      global tab_cer_app_g =      [p[0,0,0,0,0,0], p[0,0,0,0,0,0], p[0,0,0,0,0,0], p[0,0,0,0,0,0], p[0,0,0,0,0,0], p[0,0,0,0,0,0], p[0,0,0,0,0,0], p[0,0,0,0,0,0], p[0,0,0,0,0,0], p[0,0,0,0,0,0], p[0,0,0,0,0,0]]
      global tab_cer_deb_g =      [p[0,0,0,0,0,0], p[0,0,0,0,0,0], p[0,0,0,0,0,0], p[0,0,0,0,0,0], p[0,0,0,0,0,0], p[0,0,0,0,0,0], p[0,0,0,0,0,0], p[0,0,0,0,0,0], p[0,0,0,0,0,0], p[0,0,0,0,0,0], p[0,0,0,0,0,0]]
      global tab_cer_quart_g =    [p[0,0,0,0,0,0], p[0,0,0,0,0,0], p[0,0,0,0,0,0], p[0,0,0,0,0,0], p[0,0,0,0,0,0], p[0,0,0,0,0,0], p[0,0,0,0,0,0], p[0,0,0,0,0,0], p[0,0,0,0,0,0], p[0,0,0,0,0,0], p[0,0,0,0,0,0]]
      global tab_cer_mil_g =      [p[0,0,0,0,0,0], p[0,0,0,0,0,0], p[0,0,0,0,0,0], p[0,0,0,0,0,0], p[0,0,0,0,0,0], p[0,0,0,0,0,0], p[0,0,0,0,0,0], p[0,0,0,0,0,0], p[0,0,0,0,0,0], p[0,0,0,0,0,0], p[0,0,0,0,0,0]]
      global tab_cer_tro_g =      [p[0,0,0,0,0,0], p[0,0,0,0,0,0], p[0,0,0,0,0,0], p[0,0,0,0,0,0], p[0,0,0,0,0,0], p[0,0,0,0,0,0], p[0,0,0,0,0,0], p[0,0,0,0,0,0], p[0,0,0,0,0,0], p[0,0,0,0,0,0], p[0,0,0,0,0,0]]
      global tab_cer_fin_g =      [p[0,0,0,0,0,0], p[0,0,0,0,0,0], p[0,0,0,0,0,0], p[0,0,0,0,0,0], p[0,0,0,0,0,0], p[0,0,0,0,0,0], p[0,0,0,0,0,0], p[0,0,0,0,0,0], p[0,0,0,0,0,0], p[0,0,0,0,0,0], p[0,0,0,0,0,0]]
      global tab_cer_ret_g =      [p[0,0,0,0,0,0], p[0,0,0,0,0,0], p[0,0,0,0,0,0], p[0,0,0,0,0,0], p[0,0,0,0,0,0], p[0,0,0,0,0,0], p[0,0,0,0,0,0], p[0,0,0,0,0,0], p[0,0,0,0,0,0], p[0,0,0,0,0,0], p[0,0,0,0,0,0]]

       #2 nouveaux tableaux modif V2.1 (longueur 40 si 4(type)*10(nb soudures max par type) ) -> mis 45 (permettre décalage + marge)
      global tab_type_g = [0,0,0,0,0,0,0,0,0,0,0,0,0,0,0,0,0,0,0,0,0,0,0,0,0,0,0,0,0,0,0,0,0,0,0,0,0,0,0,0,0,0,0,0,0]
      global tab_job_g  = [0,0,0,0,0,0,0,0,0,0,0,0,0,0,0,0,0,0,0,0,0,0,0,0,0,0,0,0,0,0,0,0,0,0,0,0,0,0,0,0,0,0,0,0,0]

      #vitesses de soudure
      global tps_point_g = 0
      global vit_arc_g = [0,0,0,0,0,0,0,0,0,0,0]
      global vit_cer_g = [0,0,0,0,0,0,0,0,0,0,0]
      global vit_lin_g = [0,0,0,0,0,0,0,0,0,0,0]

      global nb_soud_point_g  = 0
      global nb_soud_lin_g    = 0
      global nb_soud_arc_g    = 0
      global nb_soud_cer_g    = 0

      global nbSoudure_glo_g  = 0
  end
  $ 19 "Demande"
  $ 20 "Script: demande_d.script"
  def fun_demande_d():

      close_popup()
      nb_soud_point_d = fun_demande(1)
      if (nb_soud_point_d > 0):
              tps_point_d = request_float_from_primary_client("temps des soudures points ? (s)")
      end
      nb_soud_lin_d = fun_demande(2)
      nb_soud_arc_d = fun_demande(3)
      nb_soud_cer_d = fun_demande(4)

  end
  $ 21 "Script: demande_g.script"
  def fun_demande_g():
       close_popup()
       nb_soud_point_g = fun_demande(1)
       nb_soud_lin_g = fun_demande(2)
       if nb_soud_lin_g > 0:
            vit_lin_g = fun_demande_vit(2)
       end
       nb_soud_arc_g = fun_demande(3)
       if nb_soud_arc_g > 0:
            vit_arc_g = fun_demande_vit(3)
       end
       nb_soud_cer_g = fun_demande(4)
       if nb_soud_arc_g > 0:
            vit_cer_g = fun_demande_vit(4)
       end
  end
  $ 22 "Configuration"
  $ 23 "Script: config_d.script"
  def fun_config_d():

      teach_mode()

          ################### RAZ_des_tableaux ###########################################

      fun_raz_d()

              # Init des variables de traitement
      local type = 0
      local index_soudure_point = 1
      local index_soudure_lin = 1
      local index_soudure_arc = 1
      local index_soudure_cer = 1

      local nbSoudures = 0
      local ajout = False
      close_popup()
      type = fun_demande_type_soudure()
      sync()
      while (type != 5):
          sync()
          if (type == 1):
              if (nb_soud_point_d <10):
                  ajout = True
                  fun_config_soudure_point(index_soudure_point,2) #  le ( ,2) indique la table de droite
                  index_soudure_point = index_soudure_point +1
              else:
                  ajout = False
                  popUp_tropSoudures()
              end

          elif (type == 2):
              if (nb_soud_lin_d <10):
                  ajout = True
                  fun_config_soudure_lineaire(index_soudure_lin,2)
                  index_soudure_lin = index_soudure_lin +1
              else:
                  ajout = False
                  popUp_tropSoudures()
              end

          elif (type == 3):
              if (nb_soud_arc_d <10):
                  ajout = True
                  fun_config_soudure_arc(index_soudure_arc,2)
                  index_soudure_arc = index_soudure_arc +1
              else:
                  ajout = False
                  popUp_tropSoudures()
              end

          elif (type ==4):
              if (nb_soud_cer_d <10):
                  ajout = True
                  fun_config_soudure_cercle(index_soudure_cer,2)
                  index_soudure_cer = index_soudure_cer +1
              else:
                  ajout = False
                  popUp_tropSoudures()
              end

          end

          if (ajout == True):
              tab_type_d[nbSoudures] = type
              tab_job_d[nbSoudures] = fun_demande_job(type)
              nbSoudures = nbSoudures +1
          end

          sync()
          type = fun_demande_type_soudure()
      end
      end_teach_mode()
      global nbSoudure_glo_d = nbSoudures
  end

  $ 24 "Script: config_g.script"
  def fun_config_g():

     teach_mode()

  ######################## Initialisation #######################################

      fun_raz_g()


              # Init des variables de traitement
      local type = 0
      local index_soudure_point = 1
      local index_soudure_lin = 1
      local index_soudure_arc = 1
      local index_soudure_cer = 1

      local nbSoudures = 0
      local ajout = False
      close_popup()
      type = fun_demande_type_soudure()
      sync()
      while (type != 5):
          sync()
          if (type == 1):
              if (nb_soud_point_g <10):
                  ajout = True
                  fun_config_soudure_point(index_soudure_point,1) # ( ,1 indique la table de gauche)
                  index_soudure_point = index_soudure_point +1
              else:
                  ajout = False
                  popUp_tropSoudures()
              end

          elif (type == 2):
              if (nb_soud_lin_g <10):
                  ajout = True
                  fun_config_soudure_lineaire(index_soudure_lin,1)
                  index_soudure_lin = index_soudure_lin +1
              else:
                  ajout = False
                  popUp_tropSoudures()
              end

          elif (type == 3):
              if (nb_soud_arc_g <10):
                  ajout = True
                  fun_config_soudure_arc(index_soudure_arc,1)
                  index_soudure_arc = index_soudure_arc +1
              else:
                  ajout = False
                  popUp_tropSoudures()
              end

          elif (type ==4):
              if (nb_soud_cer_g <10):
                  ajout = True
                  fun_config_soudure_cercle(index_soudure_cer,1)
                  index_soudure_cer = index_soudure_cer +1
              else:
                  ajout = False
                  popUp_tropSoudures()
              end
          end

          if (ajout == True):
              tab_type_g[nbSoudures] = type
              tab_job_g[nbSoudures] = fun_demande_job(type)
              nbSoudures = nbSoudures +1

          end

          sync()
          type = fun_demande_type_soudure()
      end

     end_teach_mode()
     global nbSoudure_glo_g = nbSoudures
  end
  $ 25 "Script: fun_config_soudure_arc.script"
  def fun_config_soudure_arc(index,table):
      if(table == 1):  # sur la table de gauche

          fun_popup_soud(1, 3, index)
          fun_front_up(adresse_bp_cobot)
          tab_arc_app_g[index] =  get_actual_tcp_pose() 	#Enregistrer position dans tableau d approche des soudures arc de cercle quand appui Bp_cobot
          close_popup()

          fun_popup_soud(2, 3, index)
          fun_front_up(adresse_bp_cobot)
          tab_arc_deb_g[index] =  get_actual_tcp_pose() 	#Enregistrer position dans tableau debut quand appui Bp_d
          close_popup()

          fun_popup_soud(4, 3, index)
          fun_front_up(adresse_bp_cobot)
          tab_arc_mil_g[index] =  get_actual_tcp_pose() 	#Enregistrer position dans tableau milieu quand appui Bp_cobot
          close_popup()

          fun_popup_soud(6, 3, index)
          fun_front_up(adresse_bp_cobot)
          tab_arc_fin_g[index] =  get_actual_tcp_pose() 	#Enregistrer position dans un tableau fin quand appui Bp_cobot
          close_popup()

          vit_arc_g[index] = fun_demande_vit(3)           #demande de vitesse des soudures lineaire

          fun_popup_soud(7, 3, index)
          fun_front_up(adresse_bp_cobot)
          tab_arc_ret_g[index] =  get_actual_tcp_pose() 	#Enregistrer position dans tableau retrait quand appui Bp_cobot
          close_popup()

          nb_soud_arc_g = nb_soud_arc_g +1

      else: #sur la table de droite
          fun_popup_soud(1, 3, index)
          fun_front_up(adresse_bp_cobot)
          tab_arc_app_d[index] =  get_actual_tcp_pose() 	#Enregistrer position dans tableau d approche des soudures arc de cercle quand appui Bp_cobot
          close_popup()

          fun_popup_soud(2, 3, index)
          fun_front_up(adresse_bp_cobot)
          tab_arc_deb_d[index] =  get_actual_tcp_pose() 	#Enregistrer position dans tableau debut quand appui Bp_d
          close_popup()

          fun_popup_soud(4, 3, index)
          fun_front_up(adresse_bp_cobot)
          tab_arc_mil_d[index] =  get_actual_tcp_pose() 	#Enregistrer position dans tableau milieu quand appui Bp_cobot
          close_popup()

          fun_popup_soud(6, 3, index)
          fun_front_up(adresse_bp_cobot)
          tab_arc_fin_d[index] =  get_actual_tcp_pose() 	#Enregistrer position dans un tableau fin quand appui Bp_cobot
          close_popup()

          vit_arc_d[index] = fun_demande_vit(3)           #demande de vitesse des soudures lineaire

          fun_popup_soud(7, 3, index)
          fun_front_up(adresse_bp_cobot)
          tab_arc_ret_d[index] =  get_actual_tcp_pose() 	#Enregistrer position dans tableau retrait quand appui Bp_cobot
          close_popup()

          nb_soud_arc_d = nb_soud_arc_d +1
      end
  end
  $ 26 "Script: fun_config_soudure_cercle.script"
  def fun_config_soudure_cercle(index,table):
      if(table == 1):  # sur la table de gauche

          fun_popup_soud(1, 4, index)
          fun_front_up(adresse_bp_cobot)
          tab_cer_app_g[index] =  get_actual_tcp_pose()     	#Enregistrer position dans tableau d approche des soudures arc de cercle quand appui Bp_cobot
          close_popup()

          fun_popup_soud(2, 4, index)
          fun_front_up(adresse_bp_cobot)
          tab_cer_deb_g[index] =  get_actual_tcp_pose()     	#Enregistrer position dans tableau debut quand appui Bp_cobot
          close_popup()

          fun_popup_soud(3, 4, index)
          fun_front_up(adresse_bp_cobot)
          tab_cer_quart_g[index] =  get_actual_tcp_pose()   	#Enregistrer position dans tableau d'approche des soudures arc de cercle quand appui Bp_d
          close_popup()

          fun_popup_soud(4, 4, index)
          fun_front_up(adresse_bp_cobot)
          tab_cer_mil_g[index] =  get_actual_tcp_pose()     	#Enregistrer position dans tableau milieu quand appui Bp_cobot
          close_popup()

          fun_popup_soud(5, 4, index)
          fun_front_up(adresse_bp_cobot)
          tab_cer_tro_g[index] =  get_actual_tcp_pose()     	#Enregistrer position dans tableau milieu quand appui Bp_cobot
          close_popup()

          fun_popup_soud(6, 4, index)
          fun_front_up(adresse_bp_cobot)
          tab_cer_fin_g[index] =  get_actual_tcp_pose()     	#Enregistrer position dans un tableau fin quand appui Bp_cobot
          close_popup()

          vit_cer_g[index] = fun_demande_vit(4)

          fun_popup_soud(7, 4, index)
          fun_front_up(adresse_bp_cobot)
          tab_cer_ret_g[index] =  get_actual_tcp_pose()    	#position de retrait est la meme que position d approche
          close_popup()

          nb_soud_cer_g= nb_soud_cer_g + 1
      else: #sur la table de droite

          fun_popup_soud(1, 4, index)
          fun_front_up(adresse_bp_cobot)
          tab_cer_app_d[index] =  get_actual_tcp_pose()     	#Enregistrer position dans tableau d approche des soudures arc de cercle quand appui Bp_cobot
          close_popup()

          fun_popup_soud(2, 4, index)
          fun_front_up(adresse_bp_cobot)
          tab_cer_deb_d[index] =  get_actual_tcp_pose()     	#Enregistrer position dans tableau debut quand appui Bp_cobot
          close_popup()

          fun_popup_soud(3, 4, index)
          fun_front_up(adresse_bp_cobot)
          tab_cer_quart_d[index] =  get_actual_tcp_pose()   	#Enregistrer position dans tableau d'approche des soudures arc de cercle quand appui Bp_d
          close_popup()

          fun_popup_soud(4, 4, index)
          fun_front_up(adresse_bp_cobot)
          tab_cer_mil_d[index] =  get_actual_tcp_pose()     	#Enregistrer position dans tableau milieu quand appui Bp_cobot
          close_popup()

          fun_popup_soud(5, 4, index)
          fun_front_up(adresse_bp_cobot)
          tab_cer_tro_d[index] =  get_actual_tcp_pose()     	#Enregistrer position dans tableau milieu quand appui Bp_cobot
          close_popup()

          fun_popup_soud(6, 4, index)
          fun_front_up(adresse_bp_cobot)
          tab_cer_fin_d[index] =  get_actual_tcp_pose()     	#Enregistrer position dans un tableau fin quand appui Bp_cobot
          close_popup()

          vit_cer_d[index] = fun_demande_vit(4)

          fun_popup_soud(7, 4, index)
          fun_front_up(adresse_bp_cobot)
          tab_cer_ret_d[index] =  get_actual_tcp_pose()    	#position de retrait est la meme que position d approche
          close_popup()

          nb_soud_cer_d = nb_soud_cer_d +1
      end
  end
  $ 27 "Script: fun_config_soudure_lineaire.script"
  def fun_config_soudure_lineaire(index, table):
      if(table == 1):  # sur la table de gauche

          fun_popup_soud(1, 2, index)
          fun_front_up(adresse_bp_cobot)
          tab_lin_app_g[index] =  get_actual_tcp_pose()     	#Enregistrer position dans tableau d approche des soudures lineaire quand appui Bp_cobot
          close_popup()

          fun_popup_soud(2, 2, index)
          fun_front_up(adresse_bp_cobot)
          tab_lin_deb_g[index] =  get_actual_tcp_pose()     	#Enregistrer position dans tableau debut quand appui Bp_cobot
          close_popup()

          fun_popup_soud(6, 2, index)
          fun_front_up(adresse_bp_cobot)
          tab_lin_fin_g[index] =  get_actual_tcp_pose()     	#Enregistrer position dans un tableau fin quand appui Bp_cobot
          close_popup()

          vit_lin_g[index] = fun_demande_vit(2)

          fun_popup_soud(7, 2, index)
          fun_front_up(adresse_bp_cobot)
          tab_lin_ret_g[index] =  get_actual_tcp_pose()     	#Enregistrer position dans tableau retrait quand appui Bp_cobot
          close_popup()

          nb_soud_lin_g = nb_soud_lin_g +1

      else: #sur la table de droite

          fun_popup_soud(1, 2, index)
          fun_front_up(adresse_bp_cobot)
          tab_lin_app_d[index] =  get_actual_tcp_pose()     	#Enregistrer position dans tableau d approche des soudures lineaire quand appui Bp_cobot
          close_popup()

          fun_popup_soud(2, 2, index)
          fun_front_up(adresse_bp_cobot)
          tab_lin_deb_d[index] =  get_actual_tcp_pose()     	#Enregistrer position dans tableau debut quand appui Bp_cobot
          close_popup()

          fun_popup_soud(6, 2, index)
          fun_front_up(adresse_bp_cobot)
          tab_lin_fin_d[index] =  get_actual_tcp_pose()     	#Enregistrer position dans un tableau fin quand appui Bp_cobot
          close_popup()

          vit_lin_d[index] = fun_demande_vit(2)

          fun_popup_soud(7, 2, index)
          fun_front_up(adresse_bp_cobot)
          tab_lin_ret_d[index] =  get_actual_tcp_pose()     	#Enregistrer position dans tableau retrait quand appui Bp_cobot
          close_popup()

          nb_soud_lin_d = nb_soud_lin_d +1
      end
  end
  $ 28 "Script: fun_config_soudure_point.script"
  def fun_config_soudure_point(index,table):

      if(table == 1):  # sur la table de gauche


          fun_popup_soud(1, 1, index)
          fun_front_up(adresse_bp_cobot)
          tab_point_app_g[index] =  get_actual_tcp_pose()   #Enregistrer position dans tableau d'approche des soudue points quand appui bouton
          close_popup()

          fun_popup_soud(2, 1, index)
          fun_front_up(adresse_bp_cobot)
          tab_point_deb_g[index] =  get_actual_tcp_pose()   #Enregistrer position debut quand appui bouton bp_cobot
          close_popup()

          tab_point_ret_g[index] = tab_point_app_g[index]         #point de retrait est le meme que le point d approche

          nb_soud_point_g = nb_soud_point_g +1

          if (nb_soud_point_g <= 1 ):
              tps_point_g = request_float_from_primary_client("temps des soudures points ? (s)")
          end




          sync()
      else: #sur la table de droite

          fun_popup_soud(1, 1, index)
          fun_front_up(adresse_bp_cobot)
          tab_point_app_d[index] =  get_actual_tcp_pose()   #Enregistrer position dans tableau d'approche des soudue points quand appui bouton
          close_popup()

          fun_popup_soud(2, 1, index)
          fun_front_up(adresse_bp_cobot)
          tab_point_deb_d[index] =  get_actual_tcp_pose()   #Enregistrer position debut quand appui bouton bp_cobot
          close_popup()

          tab_point_ret_d[index] = tab_point_app_d[index]         #point de retrait est le meme que le point d approche

          nb_soud_point_d = nb_soud_point_d +1

          if (nb_soud_point_d <= 1 ):
              tps_point_d = request_float_from_primary_client("temps des soudures points ? (s)")
          end


          sync()
      end
  end
  $ 29 "Script: popUp_tropSoudures.script"
  def popUp_tropSoudures():
      close_popup()
      popUp_tropSoudures = "Ajout impossible, deja 10 soudures de ce type"
      socket_open("127.0.0.1",29999,"internal") # open internal socket
      socket_send_line(popUp_tropSoudures,"internal")     #Affichage message
      socket_send_byte(10,"internal")
  end
  $ 30 "Script: valid_config_d.script"

  def fun_valid_config_d():
      #on demande la validation de la configuration

      validation_d = request_boolean_from_primary_client("Valider la configuration de la table droite ? Cliquer sur non pour effacer les paramètres.")

          if(validation_d ==True):

              popup2 = "popup La programmation de la pièce droite est terminée."
              socket_open("127.0.0.1",29999,"internal") # open internal socket
              socket_send_line(popup2,"internal")     #Affichage message
              socket_send_byte(10,"internal")
          config_d = 1

          else:
          nb_soud_point_d = 0
          nb_soud_lin_d = 0
          nb_soud_arc_d = 0
          nb_soud_cer_d = 0
          config_d = 0

          fun_raz_d()

          popup3 = "popup La programmation de la pièce droite a été effacée."
          socket_open("127.0.0.1",29999,"internal") # open internal socket
          socket_send_line(popup3,"internal")     #Affichage message
          socket_send_byte(10,"internal")
      end
  end
  $ 31 "Script: valid_config_g.script"
  def fun_valid_config_g():
  #on demande la validation de la configuration

      alidation_g = request_boolean_from_primary_client("Valider la programmation de la table gauche ? Cliquer sur non pour effacer les paramètres.")

      if(validation_g ==True):

          popup2 = "popup La programmation de la pièce gauche est terminée."
          socket_open("127.0.0.1",29999,"internal") # open internal socket
          socket_send_line(popup2,"internal")     #Affichage message
          socket_send_byte(10,"internal")
      config_g =1
      else:

      nb_soud_point_g = 0
      nb_soud_lin_g = 0
      nb_soud_arc_g = 0
      nb_soud_cer_g = 0
      config_g = 0

      fun_raz_g()


      popup3 = "popup La programmation de la pièce gauche a été effacée."
      socket_open("127.0.0.1",29999,"internal") # open internal socket
      socket_send_line(popup3,"internal")     #Affichage message
      socket_send_byte(10,"internal")

      end
  end
  $ 32 "Execution"
  $ 33 "Script: execution_d.script"
  def fun_execution_d():
      ######################## INITIALISATION #########################################
      #adressage
      adresse_bp_cobot = 2                                    #adresse cobot bp_cobot
      adresse_bp_d = 3                                        #adresse cobot bp_g
  #VARIABLES CI DESSUS UTILES ?????


      local index_soudure_point = 1
      local index_soudure_lin = 1
      local index_soudure_arc = 1
      local index_soudure_cer = 1

      close_popup()
      #config popup
      popup1 = "popup Table droite, éxécution..."
      socket_open("127.0.0.1",29999,"internal")
      socket_send_line(popup1,"internal")
      socket_send_byte(10,"internal")

      fun_deplacement_pose_inter(2)    #deplacement dans la position intermédiaire enregistrée

      local nbSoudures = nbSoudure_glo_d
      local soudureEnCours = 0 #soudure en cours
      local job = 0
      local typeSoudure = 0

      while (soudureEnCours<nbSoudures): #pour le moment début a 0 donc < (a voir si changement necessaire)
          job = tab_job_d[soudureEnCours]
          fun_commande_job(job)
          typeSoudure = tab_type_d[soudureEnCours]

          #switch de tous les types avec appel aux fonctions correspondantes
          if (typeSoudure == 1 ):
              fun_soudure_point(index_soudure_point,2) # ( , 2 pour signifier table de droite )
              #fun_soudure_point(index_soudure_point)
              index_soudure_point = index_soudure_point + 1
          elif (typeSoudure == 2 ):
              fun_soudure_lineaire(index_soudure_lin,2)
              index_soudure_lin = index_soudure_lin + 1
          elif (typeSoudure == 3 ):
              fun_soudure_arc(index_soudure_arc,2)
              index_soudure_arc = index_soudure_arc +1
          elif (typeSoudure == 4 ):
              fun_soudure_cercle(index_soudure_cercle,2)
              index_soudure_cercle = index_soudure_cercle +1
          else:
          end
          soudureEnCours = soudureEnCours +1
          sync()
      end
          #movej(anti_poq_d_1, a=1.4,v=1.1,t=0,r=0.005)
          #movej(anti_poq_d_2, a=1.4,v=1.1,t=0,r=0.005)
          movej(Point_Attente_D, a=0.8,v=1.05,t=0,r=0.005)
          movej(Point_init_D, a=0.8,v=1.05,t=0,r=0.005)
          movej(Point_avt_initD, a=0.8,v=1.05,t=0,r=0.005)
          movej(Point_init, a=0.8,v=1.05,t=0,r=0)
  end
  $ 34 "Script: execution_g.script"
  def fun_execution_g():
  ######################## INITIALISATION #######################################

  #adressage
  adresse_bp_cobot = 2                                    #adresse cobot bp_cobot
  adresse_bp_g = 2                                        #adresse cobot bp_g
  #VARIABLES CI DESSUS UTILES ?????


  local index_soudure_point = 1
  local index_soudure_lin = 1
  local index_soudure_arc = 1
  local index_soudure_cer = 1

  close_popup()
  #config popup
  #popup1 = "popup Table gauche, éxécution..."
  #socket_open("127.0.0.1",29999,"internal")
  #socket_send_line(popup1,"internal")
  #socket_send_byte(10,"internal")

  #fun_deplacement_pose_inter(1)

  local nbSoudures = nbSoudure_glo_g
  local soudureEnCours = 0 #soudure en cours
  local job = 0
  local typeSoudure = 0

  while (soudureEnCours<nbSoudures): #pour le moment début a 0 donc < (a voir si changement necessaire)
      job = tab_job_g[soudureEnCours]
      fun_commande_job(job)
      typeSoudure = tab_type_g[soudureEnCours]

      #switch de tous les types avec appel aux fonctions correspondantes
      if (typeSoudure == 1 ):
          #fun_soudure_point(index_soudure_point)
          fun_soudure_point(index_soudure_point,1) # ( , 1 pour signifier table de gauche )
          index_soudure_point = index_soudure_point + 1
      elif (typeSoudure == 2 ):
          fun_soudure_lineaire(index_soudure_lin,1)
          index_soudure_lin = index_soudure_lin + 1
      elif (typeSoudure == 3 ):
          fun_soudure_arc(index_soudure_arc,1)
          index_soudure_arc = index_soudure_arc +1
      elif (typeSoudure == 4 ):
          fun_soudure_cercle(index_soudure_cercle,1)
          index_soudure_cercle = index_soudure_cercle +1
      else:
      end
      soudureEnCours = soudureEnCours +1
      sync()
  end
      #movej(anti_Poq_g, a=1.4,v=1.1,t=0,r=0.005)
      #movej(Point_init, a=1.4,v=1.1,t=0,r=0.005)

     # movej(Point_Attente_G, a=0.8,v=1.05,t=0,r=0.005)
      #movej(Point_init_G, a=0.8,v=1.05,t=0,r=0.005)
     # movej(Point_init, a=0.8,v=1.05,t=0,r=0)

  end
  $ 35 "Script: fun_activer_soudure.script"
  def fun_activer_soudure():
      soudure_on = 1
      sleep(tps_init_soud)
      sync()
  end
  $ 36 "Script: fun_fin_soudure.script"
  def fun_fin_soudure(table):

      soudure_on = 0
      while(fin_soud == 0):
      end
      set_digital_out(table+4,False)                 #eteindre la lumiere pour dire que l'on soude plus

      #table +4 : les sorties numériques sont respectivements 5 table gauche & 6 table droite
      #le décalage permet d'écrire directement au bon endroit
      sync()

  end
  $ 37 "Script: fun_commande_job.script"
  #fonction ecriture des jobs vers rob3000
  def fun_commande_job(int):

      if (int == 0):
          set_digital_out(2,False)
          set_digital_out(3,False)


      elif(int == 1):
          set_digital_out(2,True)
          set_digital_out(3,False)

      elif(int == 2):
          set_digital_out(2,False)
          set_digital_out(3,True)

      elif(int == 3):
          set_digital_out(2,True)
          set_digital_out(3,True)

     # else:
     #     set_digital_out(2,False)
       #   set_digital_out(3,False)
      end
  end
  $ 38 "Script: fun_deplacement_pose_inter.script"
  def fun_deplacement_pose_inter(table):
      a_fun = 0.2
      v_fun = 1.1
      r_fun= 0
      t_fun = 0
      if (table == 1): #si 1 -> Table de gauche
        #  movej(pose_inter_g,a=a_fun,v=v_fun,t=t_fun,r=r_fun)
      else: #sinon table de droite
       #   movej(pose_inter_d,a=a_fun,v=v_fun,t=t_fun,r=r_fun)
      end
      sync()
  end
  $ 39 "Script: fun_soudure_arc.script"
  def fun_soudure_arc(Index,table):
      a_fun = 0.5
      v_fun = 1.1
      r_fun= 0.00
      t_fun = 0
      if (table == 1): #si 1 -> Table de gauche

          movej(tab_arc_app_g[Index],a_fun,v=v_fun,t=t_fun,r=r_fun)
          set_digital_out(5,True)                     #Allumer la lumiere pour dire que l'on soude
          movej(tab_arc_deb_g[Index],a_fun,v=v_fun,t=t_fun,r=r_fun)

          fun_activer_soudure()                        #appel de la fonction activer la soudure

          movec(tab_arc_mil_g[Index], tab_arc_fin_g[Index], a_fun,v=vit_arc_g[Index], r=0.002)

          fun_fin_soudure(1)                           #appel de la fonction désactiver la soudure

          movej(tab_arc_ret_g[Index],a=a_fun,v=v_fun,t=t_fun,r=r_fun)

          fun_deplacement_pose_inter(1)                     #appel de la fonction de déplacement en pose intermédiaire

      else: #sinon table de droite

          movej(tab_arc_app_d[Index],a_fun,v=v_fun,t=t_fun,r=r_fun)
          set_digital_out(6,True)                     #Allumer la lumiere pour dire que l'on soude
          movej(tab_arc_deb_d[Index],a_fun,v=v_fun,t=t_fun,r =r_fun)

          fun_activer_soudure()                        #appel de la fonction activer la soudure

          movec(tab_arc_mil_d[Index], tab_arc_fin_d[Index], a_fun,v=vit_arc_d[Index], r=0.002)

          fun_fin_soudure(2)                           #appel de la fonction désactiver la soudure

          movej(tab_arc_ret_d[Index],a_fun,v=v_fun,t=t_fun,r=r_fun)

          fun_deplacement_pose_inter(2)                     #appel de la fonction de déplacement en pose intermédiaire
      end
      sync()
  end
  $ 40 "Script: fun_soudure_cercle.script"
  def fun_soudure_cercle(Index,table):
      a_fun = 0.5
      v_fun = 1.1
      r_fun= 0.0
      t_fun = 0
      if (table == 1): #si 1 -> Table de gauche
          movej(tab_cer_app_g[Index],a=a_fun,v=v_fun,t=t_fun,r=r_fun)
          set_digital_out(5,True)                     #Allumer la lumiere pour dire que l'on soude
          movej(tab_cer_deb_g[Index],a=a_fun,v=v_fun,t=t_fun,r=r_fun)

          fun_activer_soudure()                        #appel de la fonction activer la soudure

          movec(tab_cer_quart_g[Index], tab_cer_mil_g[Index], a=a_fun,v=vit_cer_g[Index], r=0.002)
          movec(tab_cer_tro_g[Index], tab_cer_fin_g[Index], a=a_fun,v=vit_cer_g[Index], r=0.002)

          fun_fin_soudure(1)                           #appel de la fonction désactiver la soudure

          movej(tab_cer_ret_g[Index],a=a_fun, v=v_fun, t=t_fun, r=r_fun)

          fun_deplacement_pose_inter(1)                     #appel de la fonction de déplacement en pose intermédiaire

      else: #sinon table de droite
          movej(tab_cer_app_d[Index],a=a_fun,v=v_fun,t=t_fun,r=r_fun)
          set_digital_out(6,True)                     #Allumer la lumiere pour dire que l'on soude
          movej(tab_cer_deb_d[Index],a=a_fun,v=v_fun,t=t_fun,r=r_fun)

          fun_activer_soudure()                       #appel de la fonction activer la soudure

          movec(tab_cer_quart_d[Index], tab_cer_mil_d[Index], a=a_fun,v=vit_cer_d[Index], r=0.002)
          movec(tab_cer_tro_d[Index], tab_cer_fin_d[Index], a=a_fun, v=vit_cer_d[Index], r=0.002)

          fun_fin_soudure(2)                           #appel de la fonction désactiver la soudure

          movej(tab_cer_ret_d[Index],a=a_fun, v=v_fun, t=t_fun, r=r_fun)

          fun_deplacement_pose_inter(2)                     #appel de la fonction de déplacement en pose intermédiaire

      end
      sync()
  end
  $ 41 "Script: fun_soudure_lineaire.script"
  def fun_soudure_lineaire(Index,table):
      a_fun = 2
      v_fun = 4
      r_fun= 0.00
      t_fun = 0
      if (table == 1): #si 1 -> Table de gauche
          movej(tab_lin_app_g[Index],a=a_fun,v=v_fun,t=t_fun,r=r_fun)
          set_digital_out(5,True)                     #Allumer la lumiere pour dire que l'on soude
          movej(tab_lin_deb_g[Index],a=a_fun,v=v_fun,t=t_fun,r=r_fun)

          fun_activer_soudure()                         #appel de la fonction activer la soudure

          movel(tab_lin_fin_g[Index],a=a_fun,v=vit_lin_g[Index],t=t_fun)

          fun_fin_soudure(1)                           #appel de la fonction désactiver la soudure

          movej(tab_lin_ret_g[Index],a=a_fun,v=v_fun,t=t_fun,r=r_fun)

          fun_deplacement_pose_inter(1)                     #appel de la fonction de déplacement en pose intermédiaire


      else: #sinon table de droite

          movej(tab_lin_app_d[Index],a=a_fun,v=v_fun,t=t_fun,r=r_fun)
          set_digital_out(6,True)                     #Allumer la lumiere pour dire que l'on soude
          movej(tab_lin_deb_d[Index],a=a_fun,v=v_fun,t=t_fun,r=r_fun)

          fun_activer_soudure()                         #appel de la fonction activer la soudure

          movel(tab_lin_fin_d[Index],a=a_fun,v=vit_lin_d[Index],t=t_fun)

          fun_fin_soudure(2)                           #appel de la fonction désactiver la soudure

          movej(tab_lin_ret_d[Index],a=a_fun,v=v_fun,t=t_fun,r=r_fun)

          fun_deplacement_pose_inter(2)                     #appel de la fonction de déplacement en pose intermédiaire

      end
      sync()
  end
  $ 42 "Script: fun_soudure_point.script"
  def fun_soudure_point(Index,table):
      a_fun = 0.5
      v_fun = 1.1
      r_fun= 0.00
      t_fun = 0
      if (table == 1): #si 1 -> Table de gauche
          movej(tab_point_app_g[Index],a=a_fun,v=v_fun,t=t_fun,r= r_fun)
          set_digital_out(5,True)                     #Allumer la lumiere pour dire que l'on soude
          movej(tab_point_deb_g[Index],a=a_fun,v=v_fun,t=t_fun,r= r_fun)

          fun_activer_soudure()                         #appel de la fonction activer la soudure

          sleep(tps_point_g)                          #temps de soudure

          fun_fin_soudure(1)                           #appel de la fonction désactiver la soudure

          movej(tab_point_ret_g[Index],a=a_fun,v=v_fun,t=t_fun,r= r_fun)
          fun_deplacement_pose_inter(1)                     #appel de la fonction de déplacement en pose intermédiaire

      else: #sinon table de droite
          movej(tab_point_app_d[Index],a=a_fun,v=v_fun,t=t_fun,r= r_fun)
          set_digital_out(6,True)                     #Allumer la lumiere pour dire que l'on soude
          movej(tab_point_deb_d[Index],a=a_fun,v=v_fun,t=t_fun,r= r_fun)

          fun_activer_soudure()                         #appel de la fonction activer la soudure

          sleep(tps_point_d)                          #temps de soudure

          fun_fin_soudure(2)                           #appel de la fonction désactiver la soudure

          movej(tab_point_ret_d[Index],a=a_fun,v=v_fun,t=t_fun,r=r_fun)
          fun_deplacement_pose_inter(2)                     #appel de la fonction de déplacement en pose intermédiaire

      end
      sync()
  end
  $ 43 "Pas_A_Pas"
  $ 44 "Script: fun_ajouter_soudure.script"
  def fun_ajouter_soudure(sens,soudureEnCours, index_soudure_point, index_soudure_lin,index_soudure_arc,index_soudure_cercle,table):
      #pour le moment pas de vérif de trop de mouvements (doit etre inferiruer à 9par par type)

      if (table ==1):
          nbSoudures = nbSoudure_glo_g
      elif(table ==2):
          nbSoudures = nbSoudure_glo_d
      end
      local nbDecalage = 0
      local index = soudureEnCours
      local typeSoudure = 0
      local nb_soudure_type = 0
      typeSoudure = fun_demande_type_soudure()

      if (typeSoudure == 1):
        indexTypeSoudure = index_soudure_point
        if (table ==1):
            nb_soudure_type = nb_soud_point_g
        elif(table ==2):
            nb_soudure_type = nb_soud_point_d
        end
      elif (typeSoudure == 2):
          indexTypeSoudure = index_soudure_lin
          if (table ==1):
              nb_soudure_type = nb_soud_lin_g
          elif(table ==2):
              nb_soudure_type = nb_soud_lin_d
          end
      elif(typeSoudure == 3):
          indexTypeSoudure = index_soudure_arc
          if (table ==1):
              nb_soudure_type = nb_soud_arc_g
          elif(table ==2):
              nb_soudure_type = nb_soud_arc_d
          end
      elif(typeSoudure == 4):
          indexTypeSoudure = index_soudure_cercle
          if (table ==1):
              nb_soudure_type = nb_soud_cer_g
          elif(table ==2):
              nb_soudure_type = nb_soud_cer_d
          end
      end

      if (sens == 2):  #AJOUTER AVANT


          #pour les tableaux qui type & job
          index_tab_typejob = nbSoudures -1
          while(index_tab_typejob >= soudureEnCours ):
              if (table ==1):
                  tab_job_g[index_tab_typejob +1] = tab_job_g[index_tab_typejob]
                  tab_type_g[index_tab_typejob +1] = tab_type_g[index_tab_typejob]
              else:
                  tab_job_d[index_tab_typejob +1] = tab_job_d[index_tab_typejob]
                  tab_type_d[index_tab_typejob +1] = tab_type_d[index_tab_typejob]
              end

              index_tab_typejob = index_tab_typejob - 1
              sync()
          end

          #pour les tableaux de positions
          index_tab_pos = nb_soudure_type
          while(index_tab_pos >= nb_soudure_type ):
              fun_decaler_tableaux(index_tab_pos,typeSoudure,table)
              index_tab_pos = index_tab_pos -1
              sync()
          end

          #maintenant enregistrer les infos à l'index : soudureEnCoursType

          fun_inserer_soudure(typeSoudure, indexTypeSoudure, table)
          if (table ==1):
              tab_type_g[soudureEnCours]= typeSoudure
              tab_job_g[soudureEnCours] = fun_demande_job(typeSoudure)
          elif(table ==2):
              tab_type_d[soudureEnCours]= typeSoudure
              tab_job_d[soudureEnCours] = fun_demande_job(typeSoudure)
          end


      elif (sens ==3): #AJOUTER APRES

         #pour les tableaux qui type & job
         index_tab_typejob = nbSoudures
         while(index_tab_typejob >= soudureEnCours ):
              if (table ==1):
                  tab_job_g[index_tab_typejob +1] = tab_job_g[index_tab_typejob]
                  tab_type_g[index_tab_typejob +1] = tab_type_g[index_tab_typejob]
              else:
                  tab_job_d[index_tab_typejob +1] = tab_job_d[index_tab_typejob]
                  tab_type_d[index_tab_typejob +1] = tab_type_d[index_tab_typejob]
              end
             index_tab_typejob = index_tab_typejob - 1
             sync()
         end

         #pour les tableaux de positions
         index_tab_pos = nb_soudure_type
         while(index_tab_pos >= nb_soudure_type ):
             fun_decaler_tableaux(index_tab_pos,typeSoudure,table)
             index_tab_pos = index_tab_pos -1
             sync()
         end


         #maintenant enregistrer les infos à l'index : soudureEnCoursType
         #incrémenter la soudureEnCours type
         if (nb_soudure_type != 1): # dans le cas de la première l'incérement est deja a jour
              nb_soudure_type = nb_soudure_type +1
         end

         fun_inserer_soudure(typeSoudure, indexTypeSoudure, table)
         if (table ==1):
             tab_type_g[soudureEnCours+1]= typeSoudure
             tab_job_g[soudureEnCours+1] = fun_demande_job(typeSoudure)
         elif(table ==2):
             tab_type_d[soudureEnCours+1]= typeSoudure
             tab_job_d[soudureEnCours+1] = fun_demande_job(typeSoudure)
         end


      end

      sync()

      return typeSoudure
      end

  $ 45 "Script: fun_decaler_tableau.script"
  #type : 1=point 2=lineaire 3= arc de cercle 4=cercle

  #sens 2=avant 3=apres

  #table 1=gauche 2=droite

  def fun_decaler_tableaux( index_tab_pose,typeSoudure,table):



      if(table == 1): #table gauche

          if(typeSoudure ==1):
              tab_point_app_g[index_tab_pose +1] = tab_point_app_g[index_tab_pose]
              tab_point_deb_g[index_tab_pose +1] = tab_point_deb_g[index_tab_pose]
              tab_point_ret_g[index_tab_pose +1] = tab_point_ret_g[index_tab_pose]
          elif(typeSoudure == 2):
              tab_lin_app_g[index_tab_pose +1]   = tab_lin_app_g[index_tab_pose]
              tab_lin_deb_g[index_tab_pose +1]   = tab_lin_deb_g[index_tab_pose]
              tab_lin_fin_g[index_tab_pose +1]   = tab_lin_fin_g[index_tab_pose]
              tab_lin_ret_g[index_tab_pose +1]   = tab_lin_ret_g[index_tab_pose]
              vit_lin_g[index_tab_pose +1]       = vit_lin_g[index_tab_pose]
          elif(typeSoudure ==3):
              tab_arc_app_g[index_tab_pose +1]   = tab_arc_app_g[index_tab_pose]
              tab_arc_deb_g[index_tab_pose +1]   = tab_arc_deb_g[index_tab_pose]
              tab_arc_mil_g[index_tab_pose +1]   = tab_arc_mil_g[index_tab_pose]
              tab_arc_fin_g[index_tab_pose +1]   = tab_arc_fin_g[index_tab_pose]
              tab_arc_ret_g[index_tab_pose +1]   = tab_arc_ret_g[index_tab_pose]
              vit_arc_g[index_tab_pose +1]       = vit_arc_g[index_tab_pose]
          elif(typeSoudure ==4):
              tab_cer_app_g[index_tab_pose +1]   = tab_cer_app_g[index_tab_pose]
              tab_cer_deb_g[index_tab_pose +1]   = tab_cer_deb_g[index_tab_pose]
              tab_cer_quart_g[index_tab_pose +1] = tab_cer_quart_g[index_tab_pose]
              tab_cer_mil_g[index_tab_pose +1]   = tab_cer_mil_g[index_tab_pose]
              tab_cer_tro_g[index_tab_pose +1]   = tab_cer_tro_g[index_tab_pose]
              tab_cer_fin_g[index_tab_pose +1]   = tab_cer_fin_g[index_tab_pose]
              tab_cer_ret_g[index_tab_pose +1]   = tab_cer_ret_g[index_tab_pose]
              vit_cer_g[index_tab_pose +1]       = vit_cer_g[index_tab_pose]
          end

      elif(table == 2): #table droite


          if(typeSoudure ==1):
              tab_point_app_d[index_tab_pose +1] = tab_point_app_d[index_tab_pose]
              tab_point_deb_d[index_tab_pose +1] = tab_point_deb_d[index_tab_pose]
              tab_point_ret_d[index_tab_pose +1] = tab_point_ret_d[index_tab_pose]
          elif(typeSoudure == 2):
              tab_lin_app_d[index_tab_pose +1]   = tab_lin_app_d[index_tab_pose]
              tab_lin_deb_d[index_tab_pose +1]   = tab_lin_deb_d[index_tab_pose]
              tab_lin_fin_d[index_tab_pose +1]   = tab_lin_fin_d[index_tab_pose]
              tab_lin_ret_d[index_tab_pose +1]   = tab_lin_ret_d[index_tab_pose]
              vit_lin_d[index_tab_pose +1]       = vit_lin_d[index_tab_pose]
          elif(typeSoudure ==3):
              tab_arc_app_d[index_tab_pose +1]   = tab_arc_app_d[index_tab_pose]
              tab_arc_deb_d[index_tab_pose +1]   = tab_arc_deb_d[index_tab_pose]
              tab_arc_mil_d[index_tab_pose +1]   = tab_arc_mil_d[index_tab_pose]
              tab_arc_fin_d[index_tab_pose +1]   = tab_arc_fin_d[index_tab_pose]
              tab_arc_ret_d[index_tab_pose +1]   = tab_arc_ret_d[index_tab_pose]
              vit_arc_d[index_tab_pose +1]       = vit_arc_d[index_tab_pose]
          elif(typeSoudure ==4):
              tab_cer_app_d[index_tab_pose +1]   = tab_cer_app_d[index_tab_pose]
              tab_cer_deb_d[index_tab_pose +1]   = tab_cer_deb_d[index_tab_pose]
              tab_cer_quart_d[index_tab_pose +1] = tab_cer_quart_d[index_tab_pose]
              tab_cer_mil_d[index_tab_pose +1]   = tab_cer_mil_d[index_tab_pose]
              tab_cer_tro_d[index_tab_pose +1]   = tab_cer_tro_d[index_tab_pose]
              tab_cer_fin_d[index_tab_pose +1]   = tab_cer_fin_d[index_tab_pose]
              tab_cer_ret_d[index_tab_pose +1]   = tab_cer_ret_d[index_tab_pose]
              vit_cer_d[index_tab_pose +1]       = vit_cer_d[index_tab_pose]
          end


      end

  end
  $ 46 "Script: fun_inserer_soudure.script"
  def fun_inserer_soudure(type,index,table):
      teach_mode()
      #configurer une nouvelle soudure en fonction du type -> utiliser les fonction déjà développée
      if (type == 1):
          fun_config_soudure_point(index,table)
      elif (type == 2):
          fun_config_soudure_lineaire(index,table)
      elif (type == 3):
          fun_config_soudure_arc(index,table)
      elif (type ==4):
          fun_config_soudure_cercle(index,table)
      end
      end_teach_mode()
      sync()

  end
  $ 47 "Script: PasAPas_d.script"
  #######################################-_-#############################################
  def fun_Pas_A_Pas_d():

      global reglage_d = 0
      global attente = False
      global reconfig = 0
      close_popup()

      fun_deplacement_pose_inter(2)

      local index_soudure_point = 1
      local index_soudure_lin = 1
      local index_soudure_arc = 1
      local index_soudure_cer = 1

      local nbSoudures = nbSoudure_glo_d
      local soudureEnCours = 0 #soudure en cours
      local job = 0
      local typeSoudure = 0
      local TypeSoudureAjoutee = 0
      local effectuerSoudure = False
      local nouvelleSimulation = False

      while (soudureEnCours < nbSoudures):
          job = tab_job_d[soudureEnCours]
          fun_commande_job(job)

          typeSoudure = tab_type_d[soudureEnCours]
          ###
          # (1) PopUp demande simulation
          ###
          if (nouvelleSimulation == False):
              effectuerSoudure = fun_PopUp_PaP(soudureEnCours,typeSoudure,1) #appel de la fonction qui gère les PopUp
          end

          if ((effectuerSoudure == True) or(nouvelleSimulation == True)):
              ###
              # (2) Simuler()
              ###
              nouvelleSimulation  = False
              effectuerSoudure    = False

              #REALISATION DELA SOUDURE
              fun_deplacement_pose_inter(2)
              if (typeSoudure == 1 ):
                  fun_soudure_point(index_soudure_point,2) # ( , 2 pour signifier table de droite )
              elif (typeSoudure == 2 ):
                  fun_soudure_lineaire(index_soudure_lin,2)
              elif (typeSoudure == 3 ):
                  fun_soudure_arc(index_soudure_arc,2)
              elif (typeSoudure == 4 ):
                  fun_soudure_cercle(index_soudure_cer,2)
              else:
              end
              #FIN DE LA REALISATION DE LA SOUDURE
              sync()
          end
          ###
          # (3)PopUp demande modification
          ###
          modifierSoudure = fun_PopUp_PaP(soudureEnCours,typeSoudure,2) #appel de la fonction qui gère les PopUp

          if (modifierSoudure == True):
              ###
              # (4) Modifier()
              ###
              #fun_deplacement_pose_inter(2)
              teach_mode()

              if (typeSoudure == 1 ):
                  fun_config_soudure_point(index_soudure_point,2) # ( , 2 pour signifier table de droite )
              elif (typeSoudure == 2 ):
                  fun_config_soudure_lineaire(index_soudure_lin,2)
              elif (typeSoudure == 3 ):
                  fun_config_soudure_arc(index_soudure_arc,2)
              elif (typeSoudure == 4 ):
                  fun_config_soudure_cercle(index_soudure_cer,2)
              else:
              end
              end_teach_mode()
              sync()
          end
          # (5) PopUp demande ajout
          ###
          nouvelleSimulation = False
          ajouterSoudure = fun_PopUp_PaP(soudureEnCours,typeSoudure,3)
          if ((ajouterSoudure == 2) or (ajouterSoudure == 3)):
              ###
              # (6) Ajouter()
              ###
              TypeSoudureAjoutee = fun_ajouter_soudure(ajouterSoudure, soudureEnCours,index_soudure_point,index_soudure_lin,index_soudure_arc,index_soudure_cer, 2)

              if (TypeSoudureAjoutee != 5): #5 est le code retourné s'il n'y a pas d'ajout de soudure
                  nbSoudures =  nbSoudures +1
                  nbSoudure_glo_d = nbSoudures


                  typeSoudure = tab_type_d[soudureEnCours]
                  job = tab_job_d[soudureEnCours]

                  nouvelleSimulation = fun_PopUp_PaP(soudureEnCours,typeSoudure,4)

                  sync()
              end
              sync()
          end

          if (nouvelleSimulation == True):
              ###
              #(2) refaire une simulation sur cette pièce
              ###

              # pas d'incrément pour recommencer la boucle avec cette soudure
              soudureEnCours = soudureEnCours
          else:
              soudureEnCours = soudureEnCours +1
              if (typeSoudure == 1 )  :
                  index_soudure_point =index_soudure_point +1
              elif (typeSoudure == 2 ):
                  index_soudure_lin = index_soudure_lin +1
              elif (typeSoudure == 3 ):
                  index_soudure_arc = index_soudure_arc +1
              elif (typeSoudure == 4 ):
                  index_soudure_cer = index_soudure_cer+ 1
              else:
              end

          end
          sync()
      end
      sync()
  end







  $ 48 "Script: PasAPas_g.script"
  #######################################-_-#############################################
  def fun_Pas_A_Pas_g():

      global reglage_d = 0
      global attente = False
      global reconfig = 0
      close_popup()

      fun_deplacement_pose_inter(1)

      local index_soudure_point = 1
      local index_soudure_lin = 1
      local index_soudure_arc = 1
      local index_soudure_cer = 1

      local nbSoudures = nbSoudure_glo_g
      local soudureEnCours = 0 #soudure en cours
      local job = 0
      local typeSoudure = 0
      local TypeSoudureAjoutee = 0
      local effectuerSoudure = False
      local nouvelleSimulation = False

      while (soudureEnCours < nbSoudures):
          job = tab_job_g[soudureEnCours]
          fun_commande_job(job)

          typeSoudure = tab_type_g[soudureEnCours]
          ###
          # (1) PopUp demande simulation
          ###
          if (nouvelleSimulation == False):
              effectuerSoudure = fun_PopUp_PaP(soudureEnCours,typeSoudure,1) #appel de la fonction qui gère les PopUp
          end

          if ((effectuerSoudure == True) or(nouvelleSimulation == True)):
              ###
              # (2) Simuler()
              ###
              nouvelleSimulation  = False
              effectuerSoudure    = False

              #REALISATION DELA SOUDURE
              fun_deplacement_pose_inter(1)
              if (typeSoudure == 1 ):
                  fun_soudure_point(index_soudure_point,1) # ( , 2 pour signifier table de droite )
              elif (typeSoudure == 2 ):
                  fun_soudure_lineaire(index_soudure_lin,1)
              elif (typeSoudure == 3 ):
                  fun_soudure_arc(index_soudure_arc,1)
              elif (typeSoudure == 4 ):
                  fun_soudure_cercle(index_soudure_cer,1)
              else:
              end
              #FIN DE LA REALISATION DE LA SOUDURE
              sync()
          end
          ###
          # (3)PopUp demande modification
          ###
          modifierSoudure = fun_PopUp_PaP(soudureEnCours,typeSoudure,2) #appel de la fonction qui gère les PopUp

          if (modifierSoudure == True):
              ###
              # (4) Modifier()
              ###
              fun_deplacement_pose_inter(1)
              teach_mode()

              if (typeSoudure == 1 ):
                  fun_config_soudure_point(index_soudure_point,1) # ( , 2 pour signifier table de droite )
              elif (typeSoudure == 2 ):
                  fun_config_soudure_lineaire(index_soudure_lin,1)
              elif (typeSoudure == 3 ):
                  fun_config_soudure_arc(index_soudure_arc,1)
              elif (typeSoudure == 4 ):
                  fun_config_soudure_cercle(index_soudure_cer,1)
              else:
              end
              end_teach_mode()
              sync()
          end
          # (5) PopUp demande ajout
          ###
          nouvelleSimulation = False
          ajouterSoudure = fun_PopUp_PaP(soudureEnCours,typeSoudure,3)
          if ((ajouterSoudure == 2) or (ajouterSoudure == 3)):
              ###
              # (6) Ajouter()
              ###
              TypeSoudureAjoutee = fun_ajouter_soudure(ajouterSoudure, soudureEnCours,index_soudure_point,index_soudure_lin,index_soudure_arc,index_soudure_cer, 1)

              if (TypeSoudureAjoutee != 5): #5 est le code retourné s'il n'y a pas d'ajout de soudure
                  nbSoudures =  nbSoudures +1
                  nbSoudure_glo_g = nbSoudures


                  typeSoudure = tab_type_g[soudureEnCours]
                  job = tab_job_g[soudureEnCours]

                  nouvelleSimulation = fun_PopUp_PaP(soudureEnCours,typeSoudure,4)

              sync()
          end
              sync()
          end

          if (nouvelleSimulation == True):
              ###
              #(2) refaire une simulation sur cette pièce
              ###

              # pas d'incrément pour recommencer la boucle avec cette soudure
              soudureEnCours = soudureEnCours
          else:
          soudureEnCours = soudureEnCours +1
              if (typeSoudure == 1 )  :
                  index_soudure_point =index_soudure_point +1
              elif (typeSoudure == 2 ):
                  index_soudure_lin = index_soudure_lin +1
              elif (typeSoudure == 3 ):
                  index_soudure_arc = index_soudure_arc +1
              elif (typeSoudure == 4 ):
                  index_soudure_cer = index_soudure_cer+ 1
              else:
              end

          end
          sync()
      end
      sync()
  end








  $ 49 "PopUps"
  $ 50 "Configuration"
  $ 51 "Script: popup_config.script"

  def pop_up_config():
      close_popup()
      popup3 = "popup CONFIGURATION : Aucune table de configurée."
      socket_open("127.0.0.1",29999,"internal") # open internal socket
      socket_send_line(popup3,"internal")     #Affichage message
      socket_send_byte(10,"internal")
  end
  $ 52 "Script: popup_config_d.script"
  def pop_up_config_d():
      close_popup()
      popup3 = "popup CONFIGURATION : Table droite configurée."
      socket_open("127.0.0.1",29999,"internal") # open internal socket
      socket_send_line(popup3,"internal")     #Affichage message
      socket_send_byte(10,"internal")
  end
  $ 53 "Script: popup_config_g.script"
  def pop_up_config_g():
      close_popup()
      popup3 = "popup CONFIGURATION : Table droite configurée."
      socket_open("127.0.0.1",29999,"internal") # open internal socket
      socket_send_line(popup3,"internal")     #Affichage message
      socket_send_byte(10,"internal")
  end
  $ 54 "Script: popup_config_g_et_d.script"
  def pop_up_config_g_et_d():
      close_popup()
      popup3 = "popup CONFIGURATION : Les deux tables sont configurées."
      socket_open("127.0.0.1",29999,"internal") # open internal socket
      socket_send_line(popup3,"internal")     #Affichage message
      socket_send_byte(10,"internal")
  end
  $ 55 "Execution"
  $ 56 "Script: popup_deb_exe_d.script"
  def pop_up_deb_exe_d():
      close_popup()
      popup3 = "popup Table droite, éxecution... Veillez à bien fermer la porte."
      socket_open("127.0.0.1",29999,"internal") # open internal socket
      socket_send_line(popup3,"internal")     #Affichage message
      socket_send_byte(10,"internal")
  end
  $ 57 "Script: popup_deb_exe_g.script"
  def pop_up_deb_exe_g():
      close_popup()
      popup3 = "popup Table gauche, éxecution... Veillez à bien fermer la porte."
      socket_open("127.0.0.1",29999,"internal") # open internal socket
      socket_send_line(popup3,"internal")     #Affichage message
      socket_send_byte(10,"internal")
  end
  $ 58 "Script: popup_exe.script"
  def pop_up_exe():
      close_popup()
      popup1 ="popup EXECUTION : Les deux tables sont prêtes à l'éxécution" #"popup Appuyer sur le bouton gauche ou droit pour commencer l'éxécution de la pièce sur la table associée. La gestion des modes configuration et éxécution se fait à l'aide du commutateur réglage."
      socket_open("127.0.0.1",29999,"internal") # open internal socket
      socket_send_line(popup1,"internal")     #Affichage message
      socket_send_byte(10,"internal")
  end
  $ 59 "Script: popup_exe_d.script"
  def pop_up_exe_d():
      close_popup()
      popup1 = "popup EXECUTION : Table droite prête à éxécution"#"popup Appuyer sur le bouton droit pour commencer l'éxécution de la pièce configurée. La gestion des modes configuration et éxécution se fait à l'aide du commutateur réglage."
      socket_open("127.0.0.1",29999,"internal") # open internal socket
      socket_send_line(popup1,"internal")     #Affichage message
      socket_send_byte(10,"internal")
  end
  $ 60 "Script: popup_exe_g.script"
  def pop_up_exe_g():
      close_popup()
      popup1 = "popup EXECUTION : Table gauche prête à éxécution"#"popup Appuyer sur le bouton gauche pour commencer l'éxécution de la pièce configurée. La gestion des modes configuration et éxécution se fait à l'aide du commutateur réglage."
      socket_open("127.0.0.1",29999,"internal") # open internal socket
      socket_send_line(popup1,"internal")     #Affichage message
      socket_send_byte(10,"internal")
  end
  $ 61 "Script: popup_fermer_porte.script"
  def pop_up_fermer_porte():
      close_popup()
      popup3 = "popup Fermer la porte pour éxecution."
      socket_open("127.0.0.1",29999,"internal") # open internal socket
      socket_send_line(popup3,"internal")     #Affichage message
      socket_send_byte(10,"internal")
  end
  $ 62 "Pas_A_Pas"
  $ 63 "Script: fun_PopUp_PaP.script"
  def fun_PopUp_PaP(index,type,numPopUP):
      index = index +1
      char_numeroDeSoudure = to_str(index)

      local resultat = False
      local resultat2  = 0

      if (type == 1):
  		char_soudure = "point"					#si type = 1, la demande sera sur une soudure point
  	elif (type == 2):
  		char_soudure = "lineaire"				#si type = 2, la demande sera sur une soudure linéaire
  	elif (type == 3):
  		char_soudure = "arc de cercle"			#si type = 3, la demande sera sur une soudure arc de cercle
  	elif (type == 4):
  		char_soudure = "cercle"					#si type = 4, la demande sera sur une soudure cercle
  	else :
  		char_soudure = "erreur de saisie"
  	end

      if (numPopUP == 1):
          resultat  = request_boolean_from_primary_client("Soudure numero : " + char_numeroDeSoudure + ", de type : "+ char_soudure + ". Voulez vous effectuer la soudure ?(securité desactivée) Appuyer sur non pour passer à la soudure suivante. ")
          return resultat
      elif (numPopUP ==2 ):
          resultat = request_boolean_from_primary_client("Voulez vous modifier la soudure numéro :" + char_numeroDeSoudure + " ? Appuyez sur non pour continuer")
          return resultat
      elif (numPopUP ==3 ):
          resultat2 = request_integer_from_primary_client("       1-> Point SUIVANT                     Ajouter :    2-> AVANT      3-> APRES")
          return resultat2
      elif (numPopUP ==4 ):
           esultat = request_boolean_from_primary_client("Voulez vous refaire une simulation? Appuyez sur non pour continuer.")
          return resultat
      end


  end
  $ 64 "Script: popup_reg.script"
  def pop_up_reg():
      close_popup()
      popup3 = "popup PAS_A_PAS : Aucune table n'est programmée"#"popup Appuyer sur le bouton gauche ou droite pour commencer le reglage d'une pièce sur la table associée. La gestion des modes configuration, éxécution et reglage se fait à l'aide des commutateurs superieurs."
      socket_open("127.0.0.1",29999,"internal") # open internal socket
      socket_send_line(popup3,"internal")     #Affichage message
      socket_send_byte(10,"internal")
  end
  $ 65 "Script: popup_reg_d.script"
  def pop_up_reg_d():
      close_popup()
      popup3 = "popup PAS_A_PAS : Table droite programmée"#"popup La table droite est programmée. Appuyer sur le bouton gauche ou droite pour commencer le reglage d'une pièce sur la table associée. La gestion des modes programmation, éxécution et reglage se fait à l'aide des commutateurs superieurs."
      socket_open("127.0.0.1",29999,"internal") # open internal socket
      socket_send_line(popup3,"internal")     #Affichage message
      socket_send_byte(10,"internal")
  end
  $ 66 "Script: popup_reg_g.script"
  def pop_up_reg_g():
      close_popup()
      popup3 = "popup PAS_A_PAS : Table gauche programmée"#"popup La table gauche est programmée. Appuyer sur le bouton gauche ou droite pour commencer mode pas a pas et le reglage d'une pièce sur la table associée. La gestion des modes programmation, éxécution et reglage se fait à l'aide des commutateurs superieurs."
      socket_open("127.0.0.1",29999,"internal") # open internal socket
      socket_send_line(popup3,"internal")     #Affichage message
      socket_send_byte(10,"internal")
  end
  $ 67 "Script: popup_reg_gd.script"
  def pop_up_reg_gd():
      close_popup()
      popup3 = "popup PAS_A_PAS : Les deux tables sont programmées"#"popup Les deux tables sont programmées. Appuyer sur le bouton gauche ou droite pour commencer le reglage d'une pièce sur la table associée ou passez en mode éxécution à l'aide du commutateur superieur gauche pour effectuer un ou plusieurs cycle(s) de soudure(s)."
      socket_open("127.0.0.1",29999,"internal") # open internal socket
      socket_send_line(popup3,"internal")     #Affichage message
      socket_send_byte(10,"internal")
  end
  $ 334 "Thread_1"
  thread Thread_1():
    while (True):
      $ 335 "Test_Ordre_Marche"
      $ 336 "Si Test_Ordre_Mar≟ True "
      if (Test_Ordre_Mar ==   True  ):
        $ 337 "Si config_d ≟ 1  or  config_g ≟ 1"
        if (config_d  ==  1   or   config_g  ==  1):
          $ 338 "Régler Ordre_Marche=On"
          set_standard_digital_out(0, True)
          $ 339 "Attendre: 0.5"
          sleep(0.5)
          $ 340 "Si Reponse_Ordre≟ False "
          if (get_standard_digital_in(4) ==   False  ):
            $ 341 "'Si aucune reponse n'a etait recue, arret du programme'"
            # 'Si aucune reponse n'a etait recue, arret du programme'
            $ 342 "close_popup()"
            close_popup()
            $ 343 "Pop-up: Defaut : L'Ordre marche a ete coupe ( le poste est peu-etre eteint ) "
            popup("Defaut : L'Ordre marche a ete coupe ( le poste est peu-etre eteint ) ", "Erreur", False, True, blocking=False)
            halt
          end
          $ 344 "Test_Ordre_Mar≔ False "
          global Test_Ordre_Mar=  False
          $ 345 "sync()"
          sync()
        end
      end
      $ 346 "Erreur ordre marche pendant utilisation"
      $ 347 "Si Arc_On≟ True   and Reponse_Arc≟ True  and Reponse_Ordre≟ False "
      if (get_standard_digital_out(1) ==   True     and  get_standard_digital_in(5) ==   True    and  get_standard_digital_in(4) ==   False  ):
        $ 348 "'Test pour savoir si ordre marche a ete coupe pendant utilisation'"
        # 'Test pour savoir si ordre marche a ete coupe pendant utilisation'
        $ 349 "close_popup()"
        close_popup()
        $ 350 "Pop-up: Defaut : Mise sous puissance coupee pendant la trajectoire"
        popup("Defaut : Mise sous puissance coupee pendant la trajectoire", "Erreur", False, True, blocking=False)
        halt
      end
      $ 351 "sync()"
      sync()
    end
  end
  threadId_Thread_1 = run Thread_1()
  $ 352 "Thread_2"
  thread Thread_2():
    while (True):
      $ 353 "mode_soudure"
      $ 354 "Si Mode_soudure ≟  True "
      if (get_configurable_digital_in(3)  ==    True  ):
        $ 355 "Si Mode_soudure≟ True  and soudure_on ≟ True "
        if (get_configurable_digital_in(3) ==   True    and  soudure_on  ==   True  ):
          $ 356 "fin_soud≔0"
          global fin_soud=0
          $ 357 "Test_Ordre_Mar≔ True "
          global Test_Ordre_Mar=  True
          $ 358 "Test_Job≔ True "
          global Test_Job=  True
          $ 359 "Attendre Test_Ordre_Mar≟ False "
          while (not(Test_Ordre_Mar ==   False  )):
            sync()
          end
          $ 360 "Attendre Test_Job≟ False "
          while (not(Test_Job ==   False  )):
            sync()
          end
          $ 361 "Régler Arc_On=On"
          set_standard_digital_out(1, True)
          $ 362 "Test_Gaz≔ True "
          global Test_Gaz=  True
          $ 363 "'Test_Gaz permet de faire un appel dans le thread pour tester l'arriver gaz'"
          # 'Test_Gaz permet de faire un appel dans le thread pour tester l'arriver gaz'
          $ 364 "Attendre Valide_Gaz≟ True "
          while (not(Valide_Gaz ==   True  )):
            sync()
          end
          $ 365 "'Valide_Gaz permet  de connaitre quand le traitement de l'arriver gaz est terminer ans le thread.'"
          # 'Valide_Gaz permet  de connaitre quand le traitement de l'arriver gaz est terminer ans le thread.'
        else:
          $ 366 "SinonSi Mode_soudure ≟ True  and soudure_on ≟ False "
          if (get_configurable_digital_in(3)  ==   True    and  soudure_on  ==   False  ):
            $ 367 "'Attente post debit gaz'"
            # 'Attente post debit gaz'
            $ 368 "Régler Arc_On=Off"
            set_standard_digital_out(1, False)
            $ 369 "Test_Gaz≔ False "
            global Test_Gaz=  False
            $ 370 "Boucle Reponse_Arc ≟ 1"
            while (get_standard_digital_in(5)  ==  1):
              $ 371 "fin_soud≔0"
              global fin_soud=0
              $ 372 "sync()"
              sync()
            end
            $ 373 "fin_soud≔1"
            global fin_soud=1
          end
        end
      end
      $ 374 "sync()"
      sync()
    end
  end
  threadId_Thread_2 = run Thread_2()
  $ 375 "Thread_3"
  thread Thread_3():
    while (True):
      $ 376 "led_cobot_2"
      $ 377 "Si led_cobot ≟ True "
      if (led_cobot  ==   True  ):
        $ 378 "Si valider_bp_co ≟ True "
        if (get_tool_digital_in(0)  ==   True  ):
          $ 379 "Régler TO[1]=On"
          set_tool_digital_out(1, True)
          $ 380 "Attendre: 0.25"
          sleep(0.25)
          $ 381 "Régler TO[1]=Off"
          set_tool_digital_out(1, False)
          $ 382 "Attendre: 0.25"
          sleep(0.25)
          $ 383 "Régler TO[1]=On"
          set_tool_digital_out(1, True)
          $ 384 "Attendre: 0.25"
          sleep(0.25)
          $ 385 "Régler TO[1]=Off"
          set_tool_digital_out(1, False)
          $ 386 "Attendre: 0.25"
          sleep(0.25)
          $ 387 "Régler TO[1]=On"
          set_tool_digital_out(1, True)
          $ 388 "Attendre: 0.25"
          sleep(0.25)
          $ 389 "Régler TO[1]=Off"
          set_tool_digital_out(1, False)
          $ 390 "Attendre: 0.25"
          sleep(0.25)
          $ 391 "sync()"
          sync()
        end
        $ 392 "sync()"
        sync()
      end
      $ 393 "sync()"
      sync()
      $ 394 "sync()"
      sync()
    end
  end
  threadId_Thread_3 = run Thread_3()
  $ 395 "Thread_4"
  thread Thread_4():
    while (True):
      $ 396 "led_cobot"
      $ 397 "Si led_cobot ≟ True "
      if (led_cobot  ==   True  ):
        $ 398 "Boucle led_cobot ≟  True "
        while (led_cobot  ==    True  ):
          $ 399 "Régler TO[0]=On"
          set_tool_digital_out(0, True)
          $ 400 "Attendre: 0.5"
          sleep(0.5)
          $ 401 "Régler TO[0]=Off"
          set_tool_digital_out(0, False)
          $ 402 "Attendre: 0.5"
          sleep(0.5)
          $ 403 "sync()"
          sync()
        end
        $ 404 "sync()"
        sync()
      else:
        $ 405 "Sinon" "noBreak"
        $ 406 "Régler TO[0]=Off"
        set_tool_digital_out(0, False)
        $ 407 "Régler TO[1]=Off"
        set_tool_digital_out(1, False)
      end
      $ 408 "sync()"
      sync()
    end
  end
  threadId_Thread_4 = run Thread_4()
  $ 409 "Thread_5"
  thread Thread_5():
    while (True):
      $ 410 "Test_Arc_On"
      $ 411 "Erreur gaz pendant utilisation"
      $ 412 "Timer_gaz"
      $ 413 "Si Test_Gaz≟ True "
      if (Test_Gaz ==   True  ):
        $ 414 "Attendre: 1.0"
        sleep(1.0)
        $ 415 "Boucle Reponse_Arc≟ False  and Arc_On≟ True "
        thread Thread_while_415():
          while (True):
            $ 416 "'La boucle permet d'activer le timer et tester deux condition pour les Defaults'"
            # 'La boucle permet d'activer le timer et tester deux condition pour les Defaults'
            $ 417 "timer_ret_gaz: Démarrer"
            timer_ret_gaz_is_counting = True
            $ 418 "Si timer_ret_gaz>0.5"
            global thread_flag_418=0
            thread Thread_if_418():
              $ 419 "'Le timer permet de realiser une attente '"
              # 'Le timer permet de realiser une attente '
              $ 420 "close_popup()"
              close_popup()
              $ 421 "Pop-up: Defaut : Pas de retour flux, stabilisation gaz"
              popup("Defaut : Pas de retour flux, stabilisation gaz", "Erreur", False, True, blocking=False)
              halt
              thread_flag_418 = 1
            end
            if (timer_ret_gaz>0.5):
              global thread_handler_418=run Thread_if_418()
              while (thread_flag_418 == 0):
                if not(timer_ret_gaz>0.5):
                  kill thread_handler_418
                  thread_flag_418 = 2
                else:
                  sync()
                end
              end
            else:
              thread_flag_418 = 2
            end
            if (thread_flag_418 == 2):
              $ 422 "SinonSi Reponse_Ordre≟ False "
              if (get_standard_digital_in(4) ==   False  ):
                $ 423 "'Cette condition nous permet de pouvoir tout couper ordre marche pendant la boucle.'"
                # 'Cette condition nous permet de pouvoir tout couper ordre marche pendant la boucle.'
                $ 424 "close_popup()"
                close_popup()
                $ 425 "Pop-up: Defaut : Perte retour de signal, mise sous puissance generateur"
                popup("Defaut : Perte retour de signal, mise sous puissance generateur", "Erreur", False, True, blocking=False)
                halt
              end
            end
          end
        end
        if (get_standard_digital_in(5) ==   False    and  get_standard_digital_out(1) ==   True  ):
          global thread_handler_415=run Thread_while_415()
          while (get_standard_digital_in(5) ==   False    and  get_standard_digital_out(1) ==   True  ):
            sync()
          end
          kill thread_handler_415
        end
        $ 426 "Valide_Gaz≔ True "
        global Valide_Gaz=  True
        $ 427 "timer_ret_gaz: Réinitialiser"
        timer_ret_gaz = 0
      end
      $ 428 "sync()"
      sync()
    end
  end
  threadId_Thread_5 = run Thread_5()
  $ 429 "Thread_6"
  thread Thread_6():
    while (True):
      $ 430 "Test_Job"
      $ 431 "Si Test_Job≟ True "
      if (Test_Job ==   True  ):
        $ 435 "Test_Job≔ False "
        global Test_Job=  False
      end
      $ 436 "sync()"
      sync()
    end
  end
  threadId_Thread_6 = run Thread_6()
  $ 437 "Thread_7"
  thread Thread_7():
    while (True):
      $ 438 "secu"
      $ 439 "Si SecuGaucheOk ≟  False  and secu_g ≟ 1"
      if (get_configurable_digital_in(4)  ==    False    and  secu_g  ==  1):
        $ 440 "close_popup()"
        close_popup()
        $ 441 "Pop-up: ATTENTION : Defaut carter !"
        popup("ATTENTION : Defaut carter !", "Erreur", False, True, blocking=False)
        halt
      else:
        $ 442 "SinonSi SecuDroiteOk ≟ False  and secu_d ≟ 1"
        if (get_configurable_digital_in(5)  ==   False    and  secu_d  ==  1):
          $ 443 "close_popup()"
          close_popup()
          $ 444 "Pop-up: ATTENTION : Defaut carter !"
          popup("ATTENTION : Defaut carter !", "Erreur", False, True, blocking=False)
          halt
        end
      end
      $ 445 "sync()"
      sync()
    end
  end
  threadId_Thread_7 = run Thread_7()
  $ 446 "Thread_8"
  thread Thread_8():
    while (True):
      $ 447 "bloq_soud_arret"
      $ 448 "Si Mode_soudure≟ False  and Test_Gaz ≟ True "
      if (get_configurable_digital_in(3) ==   False    and  Test_Gaz  ==   True  ):
        $ 449 "close_popup()"
        close_popup()
        $ 450 "Pop-up: Defaut : L'ordre de soudure a ete coupe pendant l'utilisation."
        popup("Defaut : L'ordre de soudure a ete coupe pendant l'utilisation.", "Erreur", False, True, blocking=False)
        halt
      end
      $ 457 "sync()"
      sync()
    end
  end
  threadId_Thread_8 = run Thread_8()
  $ 468 "Thread_10"
  thread Thread_10():
    while (True):
      $ 469 "reglage"
      $ 470 "Si safe_mode ≟ 1  and Mode_manu ≟  True "
      if (safe_mode  ==  1   and  get_configurable_digital_in(7)  ==    True  ):
        $ 471 "close_popup()"
        close_popup()
        $ 472 "Pop-up: STOP !!!!"
        popup("STOP !!!!", "Erreur", False, True, blocking=False)
        halt
      end
      $ 473 "sync()"
      sync()
      $ 474 "sync()"
      sync()
    end
  end
  threadId_Thread_10 = run Thread_10()
  while (True):
    $ 68 "Programme de robot"
    $ 87 "safe_mode≔0"
    global safe_mode=0
    $ 88 "Deplacement vers position initial"
    $ 90 "Régler Cmd_Carter_Bit1=Off"
    set_configurable_digital_out(0, False)
    $ 91 "Régler Cmd_Carter_Bit2=Off"
    set_configurable_digital_out(1, False)
    $ 92 "Boucle SecuGaucheOk≟ True  or SecuDroiteOk≟ True "
    while (get_configurable_digital_in(4) ==   True    or  get_configurable_digital_in(5) ==   True  ):
      $ 93 "sync()"
      sync()
      $ 94 "'clingottement pour signifier qu'il y  un defaut sur un des carters '"
      # 'clingottement pour signifier qu'il y  un defaut sur un des carters '
      $ 95 "Régler Dcy_Voyant=Off"
      set_standard_digital_out(4, False)
      $ 96 "Régler Led_Arret=Off"
      set_configurable_digital_out(6, False)
      $ 97 "Attendre: 0.5"
      sleep(0.5)
      $ 98 "Régler Dcy_Voyant=On"
      set_standard_digital_out(4, True)
      $ 99 "Régler Led_Arret=On"
      set_configurable_digital_out(6, True)
      $ 100 "Attendre: 0.5"
      sleep(0.5)
    end
    $ 101 "Régler Led_Arret=Off"
    set_configurable_digital_out(6, False)
    $ 102 "Régler Dcy_Voyant=Off"
    set_standard_digital_out(4, False)
    $ 103 "Attendre: 2.0"
    sleep(2.0)
    $ 104 "'etre sur de l'ouverture complete du carter '"
    # 'etre sur de l'ouverture complete du carter '
    $ 105 "DéplacementL"
    $ 106 "PointPassage_12" "breakAfter"
    movel(pose_add(get_target_tcp_pose(), pose_sub(PointPassage_12_to_p, PointPassage_12_from_p)), a=0.01, v=2.0E-4)
    $ 107 "'Pos_cobot a etait affectuer a la position init (l3)'"
    # 'Pos_cobot a etait affectuer a la position init (l3)'
    $ 108 "'Pos_cobot[2] correspond a la valeur Z de la postion init (l4)'"
    # 'Pos_cobot[2] correspond a la valeur Z de la postion init (l4)'
    $ 113 "angle_base≔get_actual_joint_positions()"
    global angle_base= get_actual_joint_positions ()
    $ 114 "Si angle_base[0] ≤0.7"
    if (angle_base[0]  <= 0.7):
      $ 115 "Si angle_base[0]≥1.6"
      if (angle_base[0] >= 1.6):
        $ 116 "Départ"
        movej([0.7376820445060732, 1.3357652919721463, -2.8533326461405863, -0.44459326684985356, 1.9245067834854124, 4.003490924835204], a=1.3962634015954636, v=1.0471975511965976)
      else:
        $ 117 "SinonSi angle_base[0]>1.6"
        if (angle_base[0]>1.6):
          $ 118 "DéplacementA"
          $ 119 "Point_init_D" "breakAfter"
          movej(Point_init_D, a=1.3962634015954636, v=1.7453292519943295)
          $ 120 "Point_avt_initD" "breakAfter"
          movej(Point_avt_initD, a=1.3962634015954636, v=1.7453292519943295)
        else:
          $ 121 "SinonSi angle_base[0]<0.7"
          if (angle_base[0]<0.7):
            $ 122 "DéplacementA"
            $ 123 "Point_init_G" "breakAfter"
            movej(Point_init_G, a=1.3962634015954636, v=1.7453292519943295)
          end
        end
      end
    else:
      $ 124 "SinonSi angle_base[0]>1.6"
      if (angle_base[0]>1.6):
        $ 125 "DéplacementA"
        $ 126 "Point_init_D" "breakAfter"
        movej(Point_init_D, a=1.3962634015954636, v=1.7453292519943295)
        $ 127 "Point_avt_initD" "breakAfter"
        movej(Point_avt_initD, a=1.3962634015954636, v=1.7453292519943295)
      else:
        $ 128 "SinonSi angle_base[0]<0.7"
        if (angle_base[0]<0.7):
          $ 129 "DéplacementA"
          $ 130 "Point_init_G" "breakAfter"
          movej(Point_init_G, a=1.3962634015954636, v=1.7453292519943295)
        end
      end
    end
    $ 131 "Départ"
    movej([0.7376820445060732, 1.3357652919721463, -2.8533326461405863, -0.44459326684985356, 1.9245067834854124, 4.003490924835204], a=1.3962634015954636, v=1.0471975511965976)
    $ 132 "angle_base≔get_actual_joint_positions()"
    global angle_base= get_actual_joint_positions ()
    $ 133 "'mode config'"
    # 'mode config'
    $ 134 "Si Mode_manu ≟ False  and config_reglage ≟ False "
    if (get_configurable_digital_in(7)  ==   False    and  get_standard_digital_in(7)  ==   False  ):
      $ 135 "Si (config_g ≟ 1)  and  (config_d ≟ 1)"
      if ((config_g  ==  1)   and   (config_d  ==  1)):
        $ 136 "pop_up_config_g_et_d()"
        pop_up_config_g_et_d()
      else:
        $ 137 "SinonSi (config_g ≟1)"
        if ((config_g  == 1)):
          $ 138 "pop_up_config_g()"
          pop_up_config_g()
        else:
          $ 139 "SinonSi config_d ≟ 1"
          if (config_d  ==  1):
            $ 140 "pop_up_config_d()"
            pop_up_config_d()
          else:
            $ 141 "SinonSi (config_g ≟ 0) and (config_d ≟ 0)"
            if ((config_g  ==  0)  and  (config_d  ==  0)):
              $ 142 "pop_up_config()"
              pop_up_config()
            end
          end
        end
      end
      $ 143 "boucle≔1"
      global boucle=1
      $ 144 "Boucle (Mode_manu ≟ False ) and (boucle ≟ 1)  and (config_reglage≟ False )"
      while ((get_configurable_digital_in(7)  ==   False  )  and  (boucle  ==  1)   and  (get_standard_digital_in(7) ==   False  )):
        $ 145 "Boucle Pret_Table_Droi≟ False  and Pret_Table_Gauc≟ False  and Mode_manu ≟  False  and config_reglage≟ False "
        thread Thread_while_145():
          while (True):
            $ 146 "Régler Voyant_Table_Ga=On"
            set_standard_digital_out(5, True)
            $ 147 "Régler Voyant_Table_Dr=Off"
            set_standard_digital_out(6, False)
            $ 148 "Attendre: 0.5"
            sleep(0.5)
            $ 149 "Régler Voyant_Table_Ga=Off"
            set_standard_digital_out(5, False)
            $ 150 "Régler Voyant_Table_Dr=On"
            set_standard_digital_out(6, True)
            $ 151 "Attendre: 0.5"
            sleep(0.5)
            $ 152 "sync()"
            sync()
          end
        end
        if (get_standard_digital_in(3) ==   False    and  get_standard_digital_in(2) ==   False    and  get_configurable_digital_in(7)  ==    False    and  get_standard_digital_in(7) ==   False  ):
          global thread_handler_145=run Thread_while_145()
          while (get_standard_digital_in(3) ==   False    and  get_standard_digital_in(2) ==   False    and  get_configurable_digital_in(7)  ==    False    and  get_standard_digital_in(7) ==   False  ):
            sync()
          end
          kill thread_handler_145
        end
        $ 153 "Si Pret_Table_Gauc ≟ True "
        if (get_standard_digital_in(2)  ==   True  ):
          $ 154 "Régler Voyant_Table_Ga=On"
          set_standard_digital_out(5, True)
          $ 155 "Régler Voyant_Table_Dr=Off"
          set_standard_digital_out(6, False)
          $ 156 "'plus de demande du nombre de point a saisir'"
          # 'plus de demande du nombre de point a saisir'
          $ 157 "DéplacementA"
          $ 158 "Point_init_G" "breakAfter"
          movej(Point_init_G, a=1.3962634015954636, v=1.0471975511965976, r=0.006)
          $ 159 "Point_Attente_G" "breakAfter"
          movej(Point_Attente_G, a=1.3962634015954636, v=1.0471975511965976, r=0.006)
          $ 160 "Point_config_g" "breakAfter"
          movej(Point_config_g, a=0.6981317007977318, v=0.5235987755982988)
          $ 161 "led_cobot≔1"
          global led_cobot=1
          $ 162 "fun_config_g()"
          fun_config_g()
          $ 163 "led_cobot≔0"
          global led_cobot=0
          $ 164 "fun_valid_config_g()"
          fun_valid_config_g()
          $ 165 "DéplacementA"
          $ 167 "Point_Attente_G" "breakAfter"
          movej(Point_Attente_G, a=1.3962634015954636, v=1.0471975511965976, r=0.006)
          $ 168 "Point_init_G" "breakAfter"
          movej(Point_init_G, a=1.3962634015954636, v=1.0471975511965976, r=0.006)
          $ 170 "Départ"
          movej([0.7376820445060732, 1.3357652919721463, -2.8533326461405863, -0.44459326684985356, 1.9245067834854124, 4.003490924835204], a=1.3962634015954636, v=1.0471975511965976)
        end
        $ 171 "Si Pret_Table_Droi ≟ True "
        if (get_standard_digital_in(3)  ==   True  ):
          $ 172 "Régler Voyant_Table_Dr=On"
          set_standard_digital_out(6, True)
          $ 173 "Régler Voyant_Table_Ga=Off"
          set_standard_digital_out(5, False)
          $ 174 "DéplacementA"
          $ 175 "Point_avt_initD" "breakAfter"
          movej(Point_avt_initD, a=1.3962634015954636, v=1.0471975511965976, r=0.006)
          $ 176 "Point_init_D" "breakAfter"
          movej(Point_init_D, a=1.3962634015954636, v=1.0471975511965976)
          $ 177 "Point_Attente_D" "breakAfter"
          movej(Point_Attente_D, a=1.3962634015954636, v=1.0471975511965976, r=0.006)
          $ 178 "Point_config_d" "breakAfter"
          movej(Point_config_d, a=0.6981317007977318, v=0.5235987755982988)
          $ 179 "led_cobot≔1"
          global led_cobot=1
          $ 180 "fun_config_d()"
          fun_config_d()
          $ 181 "led_cobot≔0"
          global led_cobot=0
          $ 182 "fun_valid_config_d()"
          fun_valid_config_d()
          $ 183 "DéplacementA"
          $ 187 "Point_Attente_D" "breakAfter"
          movej(Point_Attente_D, a=1.3962634015954636, v=1.0471975511965976, r=0.006)
          $ 188 "Point_init_D" "breakAfter"
          movej(Point_init_D, a=1.3962634015954636, v=1.0471975511965976, r=0.006)
          $ 189 "Point_avt_initD" "breakAfter"
          movej(Point_avt_initD, a=1.3962634015954636, v=1.0471975511965976, r=0.006)
          $ 190 "Départ"
          movej([0.7376820445060732, 1.3357652919721463, -2.8533326461405863, -0.44459326684985356, 1.9245067834854124, 4.003490924835204], a=1.3962634015954636, v=1.0471975511965976)
        end
      end
    end
    $ 191 "''Reg''"
    # '"Reg"'
    $ 192 "Si Mode_manu ≟ False  and config_reglage ≟ True "
    if (get_configurable_digital_in(7)  ==   False    and  get_standard_digital_in(7)  ==   True  ):
      $ 193 "Si (config_g ≟ 1)  and  (config_d ≟ 1)"
      if ((config_g  ==  1)   and   (config_d  ==  1)):
        $ 194 "pop_up_reg_gd()"
        pop_up_reg_gd()
        $ 195 "boucle≔1"
        global boucle=1
      else:
        $ 196 "SinonSi config_g ≟ 1"
        if (config_g  ==  1):
          $ 197 "pop_up_reg_gd()"
          pop_up_reg_gd()
          $ 198 "boucle≔1"
          global boucle=1
        else:
          $ 199 "SinonSi config_d ≟ 1"
          if (config_d  ==  1):
            $ 200 "pop_up_reg_d()"
            pop_up_reg_d()
            $ 201 "boucle≔1"
            global boucle=1
          else:
            $ 202 "Sinon" "noBreak"
            $ 203 "close_popup()"
            close_popup()
            $ 204 "Boucle config_reglage ≟ True "
            while (get_standard_digital_in(7)  ==   True  ):
              $ 205 "Pop-up: Aucune configuration n'est actuellement detectée."
              popup("Aucune configuration n'est actuellement detectée.", "Erreur", False, True, blocking=True)
            end
          end
        end
      end
      $ 206 "boucle≔1"
      global boucle=1
      $ 207 "Boucle (Mode_manu ≟ False ) and (boucle ≟ 1)  and (config_reglage≟ True )"
      while ((get_configurable_digital_in(7)  ==   False  )  and  (boucle  ==  1)   and  (get_standard_digital_in(7) ==   True  )):
        $ 208 "Boucle Pret_Table_Droi≟ False  and Pret_Table_Gauc≟ False  and Mode_manu ≟  False  and config_reglage ≟ True "
        thread Thread_while_208():
          while (True):
            $ 209 "Si config_g ≟ 1"
            if (config_g  ==  1):
              $ 210 "Régler Voyant_Table_Ga=On"
              set_standard_digital_out(5, True)
            end
            $ 211 "Si config_d ≟ 1"
            if (config_d  ==  1):
              $ 212 "Régler Voyant_Table_Dr=On"
              set_standard_digital_out(6, True)
            end
            $ 213 "Attendre: 0.5"
            sleep(0.5)
            $ 214 "Régler Voyant_Table_Ga=Off"
            set_standard_digital_out(5, False)
            $ 215 "Régler Voyant_Table_Dr=Off"
            set_standard_digital_out(6, False)
            $ 216 "Attendre: 0.5"
            sleep(0.5)
          end
        end
        if (get_standard_digital_in(3) ==   False    and  get_standard_digital_in(2) ==   False    and  get_configurable_digital_in(7)  ==    False    and  get_standard_digital_in(7)  ==   True  ):
          global thread_handler_208=run Thread_while_208()
          while (get_standard_digital_in(3) ==   False    and  get_standard_digital_in(2) ==   False    and  get_configurable_digital_in(7)  ==    False    and  get_standard_digital_in(7)  ==   True  ):
            sync()
          end
          kill thread_handler_208
        end
        $ 217 "Si Pret_Table_Gauc ≟ True "
        if (get_standard_digital_in(2)  ==   True  ):
          $ 218 "safe_mode≔1"
          global safe_mode=1
          $ 219 "Régler Voyant_Table_Ga=On"
          set_standard_digital_out(5, True)
          $ 220 "Régler Voyant_Table_Dr=Off"
          set_standard_digital_out(6, False)
          $ 221 "DéplacementA"
          $ 222 "Point_init_G" "breakAfter"
          movej(Point_init_G, a=1.3962634015954636, v=1.0471975511965976, r=0.006)
          $ 223 "Point_Attente_G" "breakAfter"
          movej(Point_Attente_G, a=1.3962634015954636, v=1.0471975511965976, r=0.006)
          $ 224 "pose_inter_g" "breakAfter"
          movej(pose_inter_g, a=0.6981317007977318, v=0.5235987755982988)
          $ 225 "led_cobot≔1"
          global led_cobot=1
          $ 226 "fun_Pas_A_Pas_g()"
          fun_Pas_A_Pas_g()
          $ 227 "led_cobot≔0"
          global led_cobot=0
          $ 228 "safe_mode≔0"
          global safe_mode=0
          $ 229 "boucle≔0"
          global boucle=0
        end
        $ 230 "Si Pret_Table_Droi ≟ True "
        if (get_standard_digital_in(3)  ==   True  ):
          $ 231 "safe_mode≔1"
          global safe_mode=1
          $ 232 "Régler Voyant_Table_Dr=On"
          set_standard_digital_out(6, True)
          $ 233 "Régler Voyant_Table_Ga=Off"
          set_standard_digital_out(5, False)
          $ 234 "DéplacementA"
          $ 235 "Point_avt_initD" "breakAfter"
          movej(Point_avt_initD, a=1.3962634015954636, v=1.0471975511965976, r=0.006)
          $ 236 "Point_init_D" "breakAfter"
          movej(Point_init_D, a=1.3962634015954636, v=1.0471975511965976, r=0.006)
          $ 237 "pose_inter_d" "breakAfter"
          movej(pose_inter_d, a=0.6981317007977318, v=0.5235987755982988)
          $ 238 "led_cobot≔1"
          global led_cobot=1
          $ 239 "fun_Pas_A_Pas_d()"
          fun_Pas_A_Pas_d()
          $ 240 "led_cobot≔0"
          global led_cobot=0
          $ 241 "safe_mode≔0"
          global safe_mode=0
          $ 242 "boucle≔0"
          global boucle=0
        end
      end
    end
    $ 243 "'mode exe'"
    # 'mode exe'
    $ 244 "Si Mode_manu ≟ True "
    if (get_configurable_digital_in(7)  ==   True  ):
      $ 245 "Si (config_g ≟ 1)  and  (config_d ≟ 1)"
      if ((config_g  ==  1)   and   (config_d  ==  1)):
        $ 246 "pop_up_exe()"
        pop_up_exe()
        $ 247 "boucle≔1"
        global boucle=1
      else:
        $ 248 "SinonSi config_g ≟ 1"
        if (config_g  ==  1):
          $ 249 "pop_up_exe_g()"
          pop_up_exe_g()
          $ 250 "boucle≔1"
          global boucle=1
        else:
          $ 251 "SinonSi config_d ≟ 1"
          if (config_d  ==  1):
            $ 252 "pop_up_exe_d()"
            pop_up_exe_d()
            $ 253 "boucle≔1"
            global boucle=1
          else:
            $ 254 "Sinon" "noBreak"
            $ 255 "close_popup()"
            close_popup()
            $ 256 "Boucle Mode_manu ≟ True "
            while (get_configurable_digital_in(7)  ==   True  ):
              $ 257 "Pop-up: Aucune programmation n'est actuellement detectée, veillez à programmer une pièce avant de vouloir l'éxécuter."
              popup("Aucune programmation n'est actuellement detectée, veillez à programmer une pièce avant de vouloir l'éxécuter.", "Erreur", False, True, blocking=True)
            end
          end
        end
      end
      $ 258 "Boucle ( Mode_manu ≟ True )  and (boucle ≟ 1)"
      while (( get_configurable_digital_in(7)  ==   True  )   and  (boucle  ==  1)):
        $ 259 "Boucle Pret_Table_Droi≟ False  and Pret_Table_Gauc≟ False  and Mode_manu≟ True "
        thread Thread_while_259():
          while (True):
            $ 260 "Si config_g ≟ 1"
            if (config_g  ==  1):
              $ 261 "Régler Voyant_Table_Ga=On"
              set_standard_digital_out(5, True)
            end
            $ 262 "Si config_d ≟ 1"
            if (config_d  ==  1):
              $ 263 "Régler Voyant_Table_Dr=On"
              set_standard_digital_out(6, True)
            end
            $ 264 "Attendre: 0.5"
            sleep(0.5)
            $ 265 "Régler Voyant_Table_Ga=Off"
            set_standard_digital_out(5, False)
            $ 266 "Régler Voyant_Table_Dr=Off"
            set_standard_digital_out(6, False)
            $ 267 "Attendre: 0.5"
            sleep(0.5)
          end
        end
        if (get_standard_digital_in(3) ==   False    and  get_standard_digital_in(2) ==   False    and  get_configurable_digital_in(7) ==   True  ):
          global thread_handler_259=run Thread_while_259()
          while (get_standard_digital_in(3) ==   False    and  get_standard_digital_in(2) ==   False    and  get_configurable_digital_in(7) ==   True  ):
            sync()
          end
          kill thread_handler_259
        end
        $ 268 "Si (Pret_Table_Gauc ≟ True ) and (config_g ≟ True )"
        if ((get_standard_digital_in(2)  ==   True  )  and  (config_g  ==   True  )):
          $ 269 "boucle_g≔1"
          global boucle_g=1
          $ 271 "Boucle boucle_g ≟ 1"
          while (boucle_g  ==  1):
            $ 272 "Régler Cmd_Carter_Bit1=On"
            set_configurable_digital_out(0, True)
            $ 273 "Régler Voyant_Table_Ga=On"
            set_standard_digital_out(5, True)
            $ 274 "Régler Voyant_Table_Dr=Off"
            set_standard_digital_out(6, False)
            $ 275 "Attendre: 0.25"
            sleep(0.25)
            $ 276 "Régler Voyant_Table_Ga=Off"
            set_standard_digital_out(5, False)
            $ 277 "Attendre: 0.25"
            sleep(0.25)
            $ 278 "Si SecuGaucheOk ≟  False "
            if (get_configurable_digital_in(4)  ==    False  ):
              $ 279 "Régler Voyant_Table_Ga=On"
              set_standard_digital_out(5, True)
              $ 281 "Si SecuGaucheOk ≟  False "
              if (get_configurable_digital_in(4)  ==    False  ):
                $ 282 "close_popup()"
                close_popup()
                $ 283 "Attendre SecuGaucheOk=HAUT"
                while (get_configurable_digital_in(4) == False):
                  sync()
                end
              end
            end
            $ 284 "Si SecuGaucheOk ≟  True "
            if (get_configurable_digital_in(4)  ==    True  ):
              $ 285 "secu_g≔1"
              global secu_g=1
              $ 286 "Régler Voyant_Table_Ga=On"
              set_standard_digital_out(5, True)
              $ 287 "DéplacementA"
              $ 288 "Point_init_G" "breakAfter"
              movej(Point_init_G, a=1.3962634015954636, v=1.0471975511965976, r=0.006)
              $ 290 "fun_execution_g()"
              fun_execution_g()
              $ 291 "DéplacementA"
              $ 292 "Point_Attente_G" "breakAfter"
              movej(Point_Attente_G, a=1.3962634015954636, v=1.0471975511965976, r=0.006)
              $ 293 "Point_init_G" "breakAfter"
              movej(Point_init_G, a=1.3962634015954636, v=1.0471975511965976, r=0.006)
              $ 294 "Départ"
              movej([0.7376820445060732, 1.3357652919721463, -2.8533326461405863, -0.44459326684985356, 1.9245067834854124, 4.003490924835204], a=1.3962634015954636, v=1.0471975511965976)
              $ 295 "Régler Cmd_Carter_Bit1=Off"
              set_configurable_digital_out(0, False)
              $ 296 "secu_g≔0"
              global secu_g=0
              $ 297 "boucle_g≔0"
              global boucle_g=0
            end
          end
          $ 298 "boucle≔0"
          global boucle=0
        else:
          $ 299 "SinonSi (Pret_Table_Gauc ≟ True ) and (config_g ≟ False )"
          if ((get_standard_digital_in(2)  ==   True  )  and  (config_g  ==   False  )):
            $ 300 "close_popup()"
            close_popup()
            $ 301 "Pop-up: Aucune programmation n'est actuellement detectée sur la table gauche, veillez à programmer une pièce avant de vouloir l'éxécuter."
            popup("Aucune programmation n'est actuellement detectée sur la table gauche, veillez à programmer une pièce avant de vouloir l'éxécuter.", "Erreur", False, True, blocking=True)
            $ 302 "boucle≔0"
            global boucle=0
          end
        end
        $ 303 "Si (Pret_Table_Droi ≟ True ) and (config_d ≟ True )"
        if ((get_standard_digital_in(3)  ==   True  )  and  (config_d  ==   True  )):
          $ 304 "boucle_d≔1"
          global boucle_d=1
          $ 305 "pop_up_deb_exe_d()"
          pop_up_deb_exe_d()
          $ 306 "Boucle boucle_d ≟ 1"
          while (boucle_d  ==  1):
            $ 307 "Régler Cmd_Carter_Bit2=On"
            set_configurable_digital_out(1, True)
            $ 308 "Régler Voyant_Table_Ga=Off"
            set_standard_digital_out(5, False)
            $ 309 "Régler Voyant_Table_Dr=On"
            set_standard_digital_out(6, True)
            $ 310 "Attendre: 0.25"
            sleep(0.25)
            $ 311 "Régler Voyant_Table_Dr=Off"
            set_standard_digital_out(6, False)
            $ 312 "Attendre: 0.25"
            sleep(0.25)
            $ 313 "Si SecuDroiteOk ≟  False "
            if (get_configurable_digital_in(5)  ==    False  ):
              $ 314 "Régler Voyant_Table_Dr=On"
              set_standard_digital_out(6, True)
              $ 315 "Attendre: 6.0"
              sleep(6.0)
              $ 316 "Si SecuDroiteOk ≟  False "
              if (get_configurable_digital_in(5)  ==    False  ):
                $ 317 "close_popup()"
                close_popup()
                $ 318 "Attendre SecuDroiteOk=HAUT"
                while (get_configurable_digital_in(5) == False):
                  sync()
                end
              end
            end
            $ 319 "Si SecuDroiteOk ≟  True "
            if (get_configurable_digital_in(5)  ==    True  ):
              $ 320 "secu_d≔1"
              global secu_d=1
              $ 321 "Régler Voyant_Table_Dr=On"
              set_standard_digital_out(6, True)
              $ 322 "DéplacementA"
              $ 323 "Point_avt_initD" "breakAfter"
              movej(Point_avt_initD, a=1.3962634015954636, v=1.0471975511965976)
              $ 325 "fun_execution_d()"
              fun_execution_d()
              $ 326 "Régler Cmd_Carter_Bit2=Off"
              set_configurable_digital_out(1, False)
              $ 327 "secu_d≔0"
              global secu_d=0
              $ 328 "boucle_d≔0"
              global boucle_d=0
            end
          end
          $ 329 "boucle≔0"
          global boucle=0
        else:
          $ 330 "SinonSi (Pret_Table_Droi ≟ True ) and (config_d ≟ False )"
          if ((get_standard_digital_in(3)  ==   True  )  and  (config_d  ==   False  )):
            $ 331 "close_popup()"
            close_popup()
            $ 332 "Pop-up: Aucune programmation n'est actuellement detectée sur la table droite, veillez à programmer une pièce avant de vouloir l'éxécuter."
            popup("Aucune programmation n'est actuellement detectée sur la table droite, veillez à programmer une pièce avant de vouloir l'éxécuter.", "Erreur", False, True, blocking=True)
            $ 333 "boucle≔0"
            global boucle=0
          end
        end
      end
    end
  end
end
